LIN {X 0,Y 467.628,Z 314.863,A -85,B 0,C 180,E1 -7719.778,E2 -7719.778} C_VEL
LIN {X 0,Y 467.666,Z 315.024,A -85,B 0,C 180,E1 -7721.055,E2 -7721.055} C_VEL
LIN {X 0,Y 467.97,Z 316.246,A -85,B 0,C 180,E1 -7721.229,E2 -7721.229} C_VEL
LIN {X 0,Y 471.79,Z 327.707,A -85,B 0,C 180,E1 -7721.995,E2 -7721.995} C_VEL
LIN {X 0,Y 471.969,Z 329.737,A -85,B 0,C 180,E1 -7722.115,E2 -7722.115} C_VEL
LIN {X 0,Y 471.397,Z 342.99,A -85,B 0,C 180,E1 -7722.946,E2 -7722.946} C_VEL
LIN {X 0,Y 470.84,Z 354.59,A -85,B 0,C 180,E1 -7723.859,E2 -7723.859} C_VEL
LIN {X 0,Y 470.267,Z 365.932,A -85,B 0,C 180,E1 -7724.95,E2 -7724.95} C_VEL
LIN {X 0,Y 469.698,Z 376.183,A -85,B 0,C 180,E1 -7726.149,E2 -7726.149} C_VEL
LIN {X 0,Y 469.111,Z 385.408,A -85,B 0,C 180,E1 -7727.454,E2 -7727.454} C_VEL
LIN {X 0,Y 468.626,Z 393.041,A -85,B 0,C 180,E1 -7728.758,E2 -7728.758} C_VEL
LIN {X 0,Y 468.253,Z 399.346,A -85,B 0,C 180,E1 -7730.061,E2 -7730.061} C_VEL
LIN {X 0,Y 467.999,Z 404.53,A -85,B 0,C 180,E1 -7731.363,E2 -7731.363} C_VEL
LIN {X 0,Y 467.681,Z 409.923,A -85,B 0,C 180,E1 -7733.095,E2 -7733.095} C_VEL
LIN {X 0,Y 467.396,Z 413.789,A -85,B 0,C 180,E1 -7734.824,E2 -7734.824} C_VEL
LIN {X 0,Y 467.262,Z 416.221,A -85,B 0,C 180,E1 -7736.551,E2 -7736.551} C_VEL
LIN {X 0,Y 467.217,Z 417.297,A -85,B 0,C 180,E1 -7738.276,E2 -7738.276} C_VEL
LIN {X 0,Y 467.122,Z 417.057,A -85,B 0,C 180,E1 -7740,E2 -7740} C_VEL
LIN {X 0,Y 467.22,Z 415.477,A -85,B 0,C 180,E1 -7741.724,E2 -7741.724} C_VEL
LIN {X 0,Y 467.263,Z 412.569,A -85,B 0,C 180,E1 -7743.449,E2 -7743.449} C_VEL
LIN {X 0,Y 467.443,Z 408.228,A -85,B 0,C 180,E1 -7745.176,E2 -7745.176} C_VEL
LIN {X 0,Y 467.782,Z 402.317,A -85,B 0,C 180,E1 -7746.903,E2 -7746.903} C_VEL
LIN {X 0,Y 468.029,Z 395.693,A -85,B 0,C 180,E1 -7748.419,E2 -7748.419} C_VEL
LIN {X 0,Y 468.54,Z 387.434,A -85,B 0,C 180,E1 -7749.933,E2 -7749.933} C_VEL
LIN {X 0,Y 468.977,Z 378.822,A -85,B 0,C 180,E1 -7751.234,E2 -7751.234} C_VEL
LIN {X 0,Y 469.446,Z 370.309,A -85,B 0,C 180,E1 -7752.318,E2 -7752.318} C_VEL
LIN {X 0,Y 470.046,Z 358.967,A -85,B 0,C 180,E1 -7753.521,E2 -7753.521} C_VEL
LIN {X 0,Y 470.599,Z 346.534,A -85,B 0,C 180,E1 -7754.597,E2 -7754.597} C_VEL
LIN {X 0,Y 471.163,Z 334.137,A -85,B 0,C 180,E1 -7755.464,E2 -7755.464} C_VEL
LIN {X 0,Y 471.422,Z 327.577,A -85,B 0,C 180,E1 -7755.851,E2 -7755.851} C_VEL
LIN {X 0,Y 467.73,Z 315.529,A -85,B 0,C 180,E1 -7756.645,E2 -7756.645} C_VEL
LIN {X 0,Y 467.622,Z 314.897,A -85,B 0,C 180,E1 -7756.817,E2 -7756.817} C_VEL
LIN {X 0,Y 467.628,Z 314.862,A -85,B 0,C 180,E1 -7759.308,E2 -7759.308} C_VEL
LIN {X 0,Y 467.539,Z 314.87,A -85,B 0,C 180,E1 -7762.074,E2 -7762.074} C_VEL
LIN {X 0,Y 467.607,Z 314.864,A -85,B 0,C 180,E1 -7764.887,E2 -7764.887} C_VEL
LIN {X 0,Y 467.625,Z 314.856,A -85,B 0,C 180,E1 -7767.769,E2 -7767.769} C_VEL
LIN {X 0,Y 467.573,Z 314.865,A -85,B 0,C 180,E1 -7771.045,E2 -7771.045} C_VEL
LIN {X 0,Y 467.595,Z 314.863,A -85,B 0,C 180,E1 -7774.243,E2 -7774.243} C_VEL
LIN {X 0,Y 467.555,Z 314.866,A -85,B 0,C 180,E1 -7777.187,E2 -7777.187} C_VEL
LIN {X 0,Y 467.58,Z 314.867,A -85,B 0,C 180,E1 -7780.265,E2 -7780.265} C_VEL
LIN {X 0,Y 467.592,Z 314.867,A -85,B 0,C 180,E1 -7782.567,E2 -7782.567} C_VEL
LIN {X 0,Y 467.576,Z 314.863,A -85,B 0,C 180,E1 -7785.053,E2 -7785.053} C_VEL
LIN {X 0,Y 467.594,Z 314.86,A -85,B 0,C 180,E1 -7787.44,E2 -7787.44} C_VEL
LIN {X 0,Y 467.588,Z 314.863,A -85,B 0,C 180,E1 -7790.855,E2 -7790.855} C_VEL
LIN {X 0,Y 467.565,Z 314.872,A -85,B 0,C 180,E1 -7794.261,E2 -7794.261} C_VEL
LIN {X 0,Y 467.588,Z 314.861,A -85,B 0,C 180,E1 -7797.321,E2 -7797.321} C_VEL
LIN {X 0,Y 467.576,Z 314.864,A -85,B 0,C 180,E1 -7800.667,E2 -7800.667} C_VEL
LIN {X 0,Y 467.619,Z 314.857,A -85,B 0,C 180,E1 -7803.199,E2 -7803.199} C_VEL
LIN {X 0,Y 467.597,Z 314.863,A -85,B 0,C 180,E1 -7806.468,E2 -7806.468} C_VEL
LIN {X 0,Y 467.629,Z 314.86,A -85,B 0,C 180,E1 -7809.777,E2 -7809.777} C_VEL
LIN {X 0,Y 467.618,Z 314.857,A -85,B 0,C 180,E1 -7810.433,E2 -7810.433} C_VEL
LIN {X 0,Y 466.981,Z 314.938,A -85,B 0,C 180,E1 -7811.152,E2 -7811.152} C_VEL
LIN {X 0,Y 464.166,Z 315.296,A -85,B 0,C 180,E1 -7812.319,E2 -7812.319} C_VEL
LIN {X 0,Y 461.754,Z 315.599,A -85,B 0,C 180,E1 -7813.26,E2 -7813.26} C_VEL
LIN {X 0,Y 460.693,Z 315.728,A -85,B 0,C 180,E1 -7813.987,E2 -7813.987} C_VEL
LIN {X 0,Y 460.594,Z 315.737,A -85,B 0,C 180,E1 -7814.233,E2 -7814.233} C_VEL
LIN {X 0,Y 460.615,Z 315.734,A -85,B 0,C 180,E1 -7817.665,E2 -7817.665} C_VEL
LIN {X 0,Y 460.633,Z 315.728,A -85,B 0,C 180,E1 -7821.223,E2 -7821.223} C_VEL
LIN {X 0,Y 460.707,Z 315.726,A -85,B 0,C 180,E1 -7823.869,E2 -7823.869} C_VEL
LIN {X 0,Y 460.805,Z 315.708,A -85,B 0,C 180,E1 -7827.377,E2 -7827.377} C_VEL
LIN {X 0,Y 460.858,Z 315.704,A -85,B 0,C 180,E1 -7829.999,E2 -7829.999} C_VEL
LIN {X 0,Y 460.805,Z 315.706,A -85,B 0,C 180,E1 -7832.622,E2 -7832.622} C_VEL
LIN {X 0,Y 460.714,Z 315.719,A -85,B 0,C 180,E1 -7836.129,E2 -7836.129} C_VEL
LIN {X 0,Y 460.633,Z 315.727,A -85,B 0,C 180,E1 -7838.775,E2 -7838.775} C_VEL
LIN {X 0,Y 460.617,Z 315.729,A -85,B 0,C 180,E1 -7842.444,E2 -7842.444} C_VEL
LIN {X 0,Y 460.603,Z 315.733,A -85,B 0,C 180,E1 -7845.996,E2 -7845.996} C_VEL
LIN {X 0,Y 460.574,Z 315.736,A -85,B 0,C 180,E1 -7848.901,E2 -7848.901} C_VEL
LIN {X 0,Y 460.518,Z 315.749,A -85,B 0,C 180,E1 -7851.484,E2 -7851.484} C_VEL
LIN {X 0,Y 460.544,Z 315.738,A -85,B 0,C 180,E1 -7854.331,E2 -7854.331} C_VEL
LIN {X 0,Y 460.58,Z 315.741,A -85,B 0,C 180,E1 -7857.242,E2 -7857.242} C_VEL
LIN {X 0,Y 460.511,Z 315.742,A -85,B 0,C 180,E1 -7860.239,E2 -7860.239} C_VEL
LIN {X 0,Y 460.528,Z 315.747,A -85,B 0,C 180,E1 -7863.324,E2 -7863.324} C_VEL
LIN {X 0,Y 460.475,Z 315.748,A -85,B 0,C 180,E1 -7866.528,E2 -7866.528} C_VEL
LIN {X 0,Y 460.531,Z 315.74,A -85,B 0,C 180,E1 -7869.861,E2 -7869.861} C_VEL
LIN {X 0,Y 460.514,Z 315.747,A -85,B 0,C 180,E1 -7872.9,E2 -7872.9} C_VEL
LIN {X 0,Y 460.517,Z 315.742,A -85,B 0,C 180,E1 -7875.828,E2 -7875.828} C_VEL
LIN {X 0,Y 460.527,Z 315.748,A -85,B 0,C 180,E1 -7878.988,E2 -7878.988} C_VEL
LIN {X 0,Y 460.528,Z 315.744,A -85,B 0,C 180,E1 -7881.267,E2 -7881.267} C_VEL
LIN {X 0,Y 460.509,Z 315.746,A -85,B 0,C 180,E1 -7884.554,E2 -7884.554} C_VEL
LIN {X 0,Y 460.528,Z 315.74,A -85,B 0,C 180,E1 -7887.715,E2 -7887.715} C_VEL
LIN {X 0,Y 460.543,Z 315.746,A -85,B 0,C 180,E1 -7890.769,E2 -7890.769} C_VEL
LIN {X 0,Y 460.562,Z 315.736,A -85,B 0,C 180,E1 -7893.734,E2 -7893.734} C_VEL
LIN {X 0,Y 460.54,Z 315.745,A -85,B 0,C 180,E1 -7896.623,E2 -7896.623} C_VEL
LIN {X 0,Y 460.545,Z 315.738,A -85,B 0,C 180,E1 -7899.452,E2 -7899.452} C_VEL
LIN {X 0,Y 460.553,Z 315.74,A -85,B 0,C 180,E1 -7902.23,E2 -7902.23} C_VEL
LIN {X 0,Y 460.558,Z 315.74,A -85,B 0,C 180,E1 -7904.964,E2 -7904.964} C_VEL
LIN {X 0,Y 460.604,Z 315.739,A -85,B 0,C 180,E1 -7908.559,E2 -7908.559} C_VEL
LIN {X 0,Y 460.687,Z 315.723,A -85,B 0,C 180,E1 -7912.108,E2 -7912.108} C_VEL
LIN {X 0,Y 460.691,Z 315.724,A -85,B 0,C 180,E1 -7914.748,E2 -7914.748} C_VEL
LIN {X 0,Y 460.818,Z 315.704,A -85,B 0,C 180,E1 -7917.377,E2 -7917.377} C_VEL
LIN {X 0,Y 460.845,Z 315.704,A -85,B 0,C 180,E1 -7920,E2 -7920} C_VEL
LIN {X 0,Y 460.818,Z 315.708,A -85,B 0,C 180,E1 -7922.622,E2 -7922.622} C_VEL
LIN {X 0,Y 460.702,Z 315.724,A -85,B 0,C 180,E1 -7926.13,E2 -7926.13} C_VEL
LIN {X 0,Y 460.621,Z 315.73,A -85,B 0,C 180,E1 -7928.776,E2 -7928.776} C_VEL
LIN {X 0,Y 460.626,Z 315.732,A -85,B 0,C 180,E1 -7932.457,E2 -7932.457} C_VEL
LIN {X 0,Y 460.613,Z 315.736,A -85,B 0,C 180,E1 -7936.007,E2 -7936.007} C_VEL
LIN {X 0,Y 460.561,Z 315.738,A -85,B 0,C 180,E1 -7939.616,E2 -7939.616} C_VEL
LIN {X 0,Y 460.505,Z 315.746,A -85,B 0,C 180,E1 -7942.429,E2 -7942.429} C_VEL
LIN {X 0,Y 460.56,Z 315.742,A -85,B 0,C 180,E1 -7945.802,E2 -7945.802} C_VEL
LIN {X 0,Y 460.551,Z 315.742,A -85,B 0,C 180,E1 -7948.233,E2 -7948.233} C_VEL
LIN {X 0,Y 460.518,Z 315.742,A -85,B 0,C 180,E1 -7951.284,E2 -7951.284} C_VEL
LIN {X 0,Y 460.527,Z 315.741,A -85,B 0,C 180,E1 -7954.507,E2 -7954.507} C_VEL
LIN {X 0,Y 460.524,Z 315.748,A -85,B 0,C 180,E1 -7957.621,E2 -7957.621} C_VEL
LIN {X 0,Y 460.553,Z 315.743,A -85,B 0,C 180,E1 -7960.273,E2 -7960.273} C_VEL
LIN {X 0,Y 460.494,Z 315.751,A -85,B 0,C 180,E1 -7963.376,E2 -7963.376} C_VEL
LIN {X 0,Y 460.581,Z 315.992,A -85,B 0,C 180,E1 -7965.106,E2 -7965.106} C_VEL
LIN {X 0,Y 462.621,Z 325.576,A -85,B 0,C 180,E1 -7968.107,E2 -7968.107} C_VEL
LIN {X 0,Y 464.108,Z 333.816,A -85,B 0,C 180,E1 -7970.56,E2 -7970.56} C_VEL
LIN {X 0,Y 463.807,Z 340.288,A -85,B 0,C 180,E1 -7972.33,E2 -7972.33} C_VEL
LIN {X 0,Y 462.916,Z 353.475,A -85,B 0,C 180,E1 -7975.825,E2 -7975.825} C_VEL
LIN {X 0,Y 462.307,Z 365.318,A -85,B 0,C 180,E1 -7978.879,E2 -7978.879} C_VEL
LIN {X 0,Y 461.866,Z 375.16,A -85,B 0,C 180,E1 -7981.36,E2 -7981.36} C_VEL
LIN {X 0,Y 461.397,Z 387.321,A -85,B 0,C 180,E1 -7984.365,E2 -7984.365} C_VEL
LIN {X 0,Y 461.011,Z 398.687,A -85,B 0,C 180,E1 -7987.125,E2 -7987.125} C_VEL
LIN {X 0,Y 460.583,Z 412.328,A -85,B 0,C 180,E1 -7990.386,E2 -7990.386} C_VEL
LIN {X 0,Y 460.517,Z 415.483,A -85,B 0,C 180,E1 -7991.083,E2 -7991.083} C_VEL
LIN {X 0,Y 461.15,Z 420.195,A -85,B 0,C 180,E1 -7991.244,E2 -7991.244} C_VEL
LIN {X 0,Y 462.995,Z 434.142,A -85,B 0,C 180,E1 -7991.685,E2 -7991.685} C_VEL
LIN {X 0,Y 464.3,Z 444.091,A -85,B 0,C 180,E1 -7992.094,E2 -7992.094} C_VEL
LIN {X 0,Y 463.679,Z 457.656,A -85,B 0,C 180,E1 -7992.725,E2 -7992.725} C_VEL
LIN {X 0,Y 462.956,Z 471.604,A -85,B 0,C 180,E1 -7993.577,E2 -7993.577} C_VEL
LIN {X 0,Y 462.209,Z 484.511,A -85,B 0,C 180,E1 -7994.569,E2 -7994.569} C_VEL
LIN {X 0,Y 461.577,Z 496.243,A -85,B 0,C 180,E1 -7995.676,E2 -7995.676} C_VEL
LIN {X 0,Y 460.939,Z 507.823,A -85,B 0,C 180,E1 -7997.004,E2 -7997.004} C_VEL
LIN {X 0,Y 460.56,Z 517.359,A -85,B 0,C 180,E1 -7998.336,E2 -7998.336} C_VEL
LIN {X 0,Y 460.142,Z 526.442,A -85,B 0,C 180,E1 -7999.885,E2 -7999.885} C_VEL
LIN {X 0,Y 459.972,Z 532.875,A -85,B 0,C 180,E1 -8001.212,E2 -8001.212} C_VEL
LIN {X 0,Y 459.892,Z 538.158,A -85,B 0,C 180,E1 -8002.537,E2 -8002.537} C_VEL
LIN {X 0,Y 459.93,Z 542.435,A -85,B 0,C 180,E1 -8003.861,E2 -8003.861} C_VEL
LIN {X 0,Y 459.886,Z 546.709,A -85,B 0,C 180,E1 -8005.619,E2 -8005.619} C_VEL
LIN {X 0,Y 459.897,Z 549.469,A -85,B 0,C 180,E1 -8007.373,E2 -8007.373} C_VEL
LIN {X 0,Y 459.864,Z 550.771,A -85,B 0,C 180,E1 -8009.125,E2 -8009.125} C_VEL
LIN {X 0,Y 459.999,Z 550.906,A -85,B 0,C 180,E1 -8010.001,E2 -8010.001} C_VEL
LIN {X 0,Y 460.019,Z 550.665,A -85,B 0,C 180,E1 -8010.876,E2 -8010.876} C_VEL
LIN {X 0,Y 459.945,Z 549.078,A -85,B 0,C 180,E1 -8012.628,E2 -8012.628} C_VEL
LIN {X 0,Y 460.043,Z 546.043,A -85,B 0,C 180,E1 -8014.382,E2 -8014.382} C_VEL
LIN {X 0,Y 459.977,Z 542.746,A -85,B 0,C 180,E1 -8015.7,E2 -8015.7} C_VEL
LIN {X 0,Y 460.012,Z 536.886,A -85,B 0,C 180,E1 -8017.462,E2 -8017.462} C_VEL
LIN {X 0,Y 460.066,Z 530.243,A -85,B 0,C 180,E1 -8019.009,E2 -8019.009} C_VEL
LIN {X 0,Y 460.301,Z 521.996,A -85,B 0,C 180,E1 -8020.558,E2 -8020.558} C_VEL
LIN {X 0,Y 460.556,Z 513.41,A -85,B 0,C 180,E1 -8021.889,E2 -8021.889} C_VEL
LIN {X 0,Y 460.958,Z 503.141,A -85,B 0,C 180,E1 -8023.221,E2 -8023.221} C_VEL
LIN {X 0,Y 461.475,Z 491.831,A -85,B 0,C 180,E1 -8024.442,E2 -8024.442} C_VEL
LIN {X 0,Y 462.189,Z 479.47,A -85,B 0,C 180,E1 -8025.546,E2 -8025.546} C_VEL
LIN {X 0,Y 462.842,Z 465.889,A -85,B 0,C 180,E1 -8026.542,E2 -8026.542} C_VEL
LIN {X 0,Y 463.548,Z 452.57,A -85,B 0,C 180,E1 -8027.319,E2 -8027.319} C_VEL
LIN {X 0,Y 463.934,Z 443.508,A -85,B 0,C 180,E1 -8027.751,E2 -8027.751} C_VEL
LIN {X 0,Y 462.67,Z 432.253,A -85,B 0,C 180,E1 -8028.259,E2 -8028.259} C_VEL
LIN {X 0,Y 461.343,Z 416.975,A -85,B 0,C 180,E1 -8028.776,E2 -8028.776} C_VEL
LIN {X 0,Y 460.379,Z 409.518,A -85,B 0,C 180,E1 -8029.018,E2 -8029.018} C_VEL
LIN {X 0,Y 460.435,Z 407.458,A -85,B 0,C 180,E1 -8029.395,E2 -8029.395} C_VEL
LIN {X 0,Y 460.579,Z 392.689,A -85,B 0,C 180,E1 -8032.662,E2 -8032.662} C_VEL
LIN {X 0,Y 460.751,Z 378.539,A -85,B 0,C 180,E1 -8035.849,E2 -8035.849} C_VEL
LIN {X 0,Y 460.983,Z 364.098,A -85,B 0,C 180,E1 -8039.201,E2 -8039.201} C_VEL
LIN {X 0,Y 461.17,Z 351.605,A -85,B 0,C 180,E1 -8042.235,E2 -8042.235} C_VEL
LIN {X 0,Y 461.757,Z 337.842,A -85,B 0,C 180,E1 -8045.8,E2 -8045.8} C_VEL
LIN {X 0,Y 462.679,Z 328.181,A -85,B 0,C 180,E1 -8048.52,E2 -8048.52} C_VEL
LIN {X 0,Y 462.076,Z 323.427,A -85,B 0,C 180,E1 -8050.069,E2 -8050.069} C_VEL
LIN {X 0,Y 460.965,Z 317.845,A -85,B 0,C 180,E1 -8052.132,E2 -8052.132} C_VEL
LIN {X 0,Y 460.532,Z 315.801,A -85,B 0,C 180,E1 -8052.999,E2 -8052.999} C_VEL
LIN {X 0,Y 460.515,Z 315.749,A -85,B 0,C 180,E1 -8055.831,E2 -8055.831} C_VEL
LIN {X 0,Y 460.542,Z 315.744,A -85,B 0,C 180,E1 -8058.99,E2 -8058.99} C_VEL
LIN {X 0,Y 460.547,Z 315.744,A -85,B 0,C 180,E1 -8061.269,E2 -8061.269} C_VEL
LIN {X 0,Y 460.517,Z 315.744,A -85,B 0,C 180,E1 -8064.555,E2 -8064.555} C_VEL
LIN {X 0,Y 460.535,Z 315.746,A -85,B 0,C 180,E1 -8067.716,E2 -8067.716} C_VEL
LIN {X 0,Y 460.543,Z 315.742,A -85,B 0,C 180,E1 -8070.769,E2 -8070.769} C_VEL
LIN {X 0,Y 460.567,Z 315.741,A -85,B 0,C 180,E1 -8073.735,E2 -8073.735} C_VEL
LIN {X 0,Y 460.55,Z 315.743,A -85,B 0,C 180,E1 -8076.624,E2 -8076.624} C_VEL
LIN {X 0,Y 460.556,Z 315.744,A -85,B 0,C 180,E1 -8079.453,E2 -8079.453} C_VEL
LIN {X 0,Y 460.633,Z 315.941,A -85,B 0,C 180,E1 -8080.733,E2 -8080.733} C_VEL
LIN {X 0,Y 460.904,Z 317.05,A -85,B 0,C 180,E1 -8080.892,E2 -8080.892} C_VEL
LIN {X 0,Y 465.016,Z 329.082,A -85,B 0,C 180,E1 -8081.724,E2 -8081.724} C_VEL
LIN {X 0,Y 465.252,Z 332.956,A -85,B 0,C 180,E1 -8081.961,E2 -8081.961} C_VEL
LIN {X 0,Y 464.64,Z 345.545,A -85,B 0,C 180,E1 -8082.791,E2 -8082.791} C_VEL
LIN {X 0,Y 464.029,Z 358.222,A -85,B 0,C 180,E1 -8083.841,E2 -8083.841} C_VEL
LIN {X 0,Y 463.39,Z 369.118,A -85,B 0,C 180,E1 -8084.946,E2 -8084.946} C_VEL
LIN {X 0,Y 462.771,Z 379.447,A -85,B 0,C 180,E1 -8086.221,E2 -8086.221} C_VEL
LIN {X 0,Y 462.228,Z 387.925,A -85,B 0,C 180,E1 -8087.487,E2 -8087.487} C_VEL
LIN {X 0,Y 461.586,Z 396.39,A -85,B 0,C 180,E1 -8089.029,E2 -8089.029} C_VEL
LIN {X 0,Y 461.197,Z 402.314,A -85,B 0,C 180,E1 -8090.35,E2 -8090.35} C_VEL
LIN {X 0,Y 460.937,Z 407.14,A -85,B 0,C 180,E1 -8091.672,E2 -8091.672} C_VEL
LIN {X 0,Y 460.681,Z 412.123,A -85,B 0,C 180,E1 -8093.43,E2 -8093.43} C_VEL
LIN {X 0,Y 460.404,Z 414.86,A -85,B 0,C 180,E1 -8094.745,E2 -8094.745} C_VEL
LIN {X 0,Y 460.25,Z 417.278,A -85,B 0,C 180,E1 -8096.498,E2 -8096.498} C_VEL
LIN {X 0,Y 460.201,Z 418.341,A -85,B 0,C 180,E1 -8098.25,E2 -8098.25} C_VEL
LIN {X 0,Y 460.1,Z 418.084,A -85,B 0,C 180,E1 -8100,E2 -8100} C_VEL
LIN {X 0,Y 460.203,Z 416.483,A -85,B 0,C 180,E1 -8101.75,E2 -8101.75} C_VEL
LIN {X 0,Y 460.244,Z 413.549,A -85,B 0,C 180,E1 -8103.502,E2 -8103.502} C_VEL
LIN {X 0,Y 460.443,Z 409.175,A -85,B 0,C 180,E1 -8105.255,E2 -8105.255} C_VEL
LIN {X 0,Y 460.806,Z 403.228,A -85,B 0,C 180,E1 -8107.009,E2 -8107.009} C_VEL
LIN {X 0,Y 461.078,Z 396.57,A -85,B 0,C 180,E1 -8108.547,E2 -8108.547} C_VEL
LIN {X 0,Y 461.612,Z 388.269,A -85,B 0,C 180,E1 -8110.084,E2 -8110.084} C_VEL
LIN {X 0,Y 462.074,Z 379.621,A -85,B 0,C 180,E1 -8111.404,E2 -8111.404} C_VEL
LIN {X 0,Y 462.574,Z 371.079,A -85,B 0,C 180,E1 -8112.504,E2 -8112.504} C_VEL
LIN {X 0,Y 463.192,Z 359.827,A -85,B 0,C 180,E1 -8113.711,E2 -8113.711} C_VEL
LIN {X 0,Y 463.728,Z 348.623,A -85,B 0,C 180,E1 -8114.706,E2 -8114.706} C_VEL
LIN {X 0,Y 464.356,Z 336.506,A -85,B 0,C 180,E1 -8115.584,E2 -8115.584} C_VEL
LIN {X 0,Y 464.596,Z 328.994,A -85,B 0,C 180,E1 -8116.045,E2 -8116.045} C_VEL
LIN {X 0,Y 460.652,Z 316.238,A -85,B 0,C 180,E1 -8116.908,E2 -8116.908} C_VEL
LIN {X 0,Y 460.591,Z 315.767,A -85,B 0,C 180,E1 -8117.082,E2 -8117.082} C_VEL
LIN {X 0,Y 460.573,Z 315.739,A -85,B 0,C 180,E1 -8119.616,E2 -8119.616} C_VEL
LIN {X 0,Y 460.515,Z 315.748,A -85,B 0,C 180,E1 -8122.429,E2 -8122.429} C_VEL
LIN {X 0,Y 460.573,Z 315.734,A -85,B 0,C 180,E1 -8125.802,E2 -8125.802} C_VEL
LIN {X 0,Y 460.557,Z 315.739,A -85,B 0,C 180,E1 -8128.233,E2 -8128.233} C_VEL
LIN {X 0,Y 460.526,Z 315.741,A -85,B 0,C 180,E1 -8131.283,E2 -8131.283} C_VEL
LIN {X 0,Y 460.539,Z 315.746,A -85,B 0,C 180,E1 -8134.506,E2 -8134.506} C_VEL
LIN {X 0,Y 460.507,Z 315.743,A -85,B 0,C 180,E1 -8137.623,E2 -8137.623} C_VEL
LIN {X 0,Y 460.544,Z 315.743,A -85,B 0,C 180,E1 -8140.269,E2 -8140.269} C_VEL
LIN {X 0,Y 460.503,Z 315.743,A -85,B 0,C 180,E1 -8143.376,E2 -8143.376} C_VEL
LIN {X 0,Y 460.515,Z 315.747,A -85,B 0,C 180,E1 -8146.626,E2 -8146.626} C_VEL
LIN {X 0,Y 460.549,Z 315.739,A -85,B 0,C 180,E1 -8149.73,E2 -8149.73} C_VEL
LIN {X 0,Y 460.505,Z 315.748,A -85,B 0,C 180,E1 -8152.524,E2 -8152.524} C_VEL
LIN {X 0,Y 460.552,Z 315.738,A -85,B 0,C 180,E1 -8155.624,E2 -8155.624} C_VEL
LIN {X 0,Y 460.543,Z 315.74,A -85,B 0,C 180,E1 -8158.744,E2 -8158.744} C_VEL
LIN {X 0,Y 460.595,Z 315.739,A -85,B 0,C 180,E1 -8162.252,E2 -8162.252} C_VEL
LIN {X 0,Y 460.538,Z 315.741,A -85,B 0,C 180,E1 -8165.667,E2 -8165.667} C_VEL
LIN {X 0,Y 460.528,Z 315.742,A -85,B 0,C 180,E1 -8168.578,E2 -8168.578} C_VEL
LIN {X 0,Y 460.597,Z 315.732,A -85,B 0,C 180,E1 -8171.311,E2 -8171.311} C_VEL
LIN {X 0,Y 460.594,Z 315.737,A -85,B 0,C 180,E1 -8174.233,E2 -8174.233} C_VEL
LIN {X 0,Y 459.892,Z 315.82,A -85,B 0,C 180,E1 -8174.963,E2 -8174.963} C_VEL
LIN {X 0,Y 457.031,Z 316.181,A -85,B 0,C 180,E1 -8176.148,E2 -8176.148} C_VEL
LIN {X 0,Y 454.642,Z 316.476,A -85,B 0,C 180,E1 -8177.104,E2 -8177.104} C_VEL
LIN {X 0,Y 453.631,Z 316.606,A -85,B 0,C 180,E1 -8177.842,E2 -8177.842} C_VEL
LIN {X 0,Y 453.555,Z 316.61,A -85,B 0,C 180,E1 -8178.092,E2 -8178.092} C_VEL
LIN {X 0,Y 453.597,Z 316.604,A -85,B 0,C 180,E1 -8181.086,E2 -8181.086} C_VEL
LIN {X 0,Y 453.675,Z 316.601,A -85,B 0,C 180,E1 -8183.774,E2 -8183.774} C_VEL
LIN {X 0,Y 453.749,Z 316.587,A -85,B 0,C 180,E1 -8187.336,E2 -8187.336} C_VEL
LIN {X 0,Y 453.828,Z 316.579,A -85,B 0,C 180,E1 -8189.999,E2 -8189.999} C_VEL
LIN {X 0,Y 453.749,Z 316.584,A -85,B 0,C 180,E1 -8192.662,E2 -8192.662} C_VEL
LIN {X 0,Y 453.682,Z 316.594,A -85,B 0,C 180,E1 -8196.224,E2 -8196.224} C_VEL
LIN {X 0,Y 453.596,Z 316.604,A -85,B 0,C 180,E1 -8198.912,E2 -8198.912} C_VEL
LIN {X 0,Y 453.567,Z 316.607,A -85,B 0,C 180,E1 -8202.528,E2 -8202.528} C_VEL
LIN {X 0,Y 453.548,Z 316.61,A -85,B 0,C 180,E1 -8206.195,E2 -8206.195} C_VEL
LIN {X 0,Y 453.523,Z 316.615,A -85,B 0,C 180,E1 -8209.04,E2 -8209.04} C_VEL
LIN {X 0,Y 453.479,Z 316.621,A -85,B 0,C 180,E1 -8211.835,E2 -8211.835} C_VEL
LIN {X 0,Y 453.515,Z 316.615,A -85,B 0,C 180,E1 -8214.733,E2 -8214.733} C_VEL
LIN {X 0,Y 453.538,Z 316.612,A -85,B 0,C 180,E1 -8217.96,E2 -8217.96} C_VEL
LIN {X 0,Y 453.467,Z 316.624,A -85,B 0,C 180,E1 -8221.524,E2 -8221.524} C_VEL
LIN {X 0,Y 453.486,Z 316.62,A -85,B 0,C 180,E1 -8224.776,E2 -8224.776} C_VEL
LIN {X 0,Y 453.463,Z 316.62,A -85,B 0,C 180,E1 -8228.31,E2 -8228.31} C_VEL
LIN {X 0,Y 453.492,Z 316.618,A -85,B 0,C 180,E1 -8230.608,E2 -8230.608} C_VEL
LIN {X 0,Y 453.461,Z 316.626,A -85,B 0,C 180,E1 -8233.244,E2 -8233.244} C_VEL
LIN {X 0,Y 453.471,Z 316.62,A -85,B 0,C 180,E1 -8235.779,E2 -8235.779} C_VEL
LIN {X 0,Y 453.49,Z 316.62,A -85,B 0,C 180,E1 -8239.39,E2 -8239.39} C_VEL
LIN {X 0,Y 453.47,Z 316.62,A -85,B 0,C 180,E1 -8242.222,E2 -8242.222} C_VEL
LIN {X 0,Y 453.484,Z 316.621,A -85,B 0,C 180,E1 -8245.221,E2 -8245.221} C_VEL
LIN {X 0,Y 453.482,Z 316.621,A -85,B 0,C 180,E1 -8248.469,E2 -8248.469} C_VEL
LIN {X 0,Y 453.51,Z 316.617,A -85,B 0,C 180,E1 -8251.288,E2 -8251.288} C_VEL
LIN {X 0,Y 453.519,Z 316.615,A -85,B 0,C 180,E1 -8254.284,E2 -8254.284} C_VEL
LIN {X 0,Y 453.474,Z 316.621,A -85,B 0,C 180,E1 -8257.203,E2 -8257.203} C_VEL
LIN {X 0,Y 453.498,Z 316.617,A -85,B 0,C 180,E1 -8260.065,E2 -8260.065} C_VEL
LIN {X 0,Y 453.5,Z 316.62,A -85,B 0,C 180,E1 -8262.875,E2 -8262.875} C_VEL
LIN {X 0,Y 453.508,Z 316.614,A -85,B 0,C 180,E1 -8265.643,E2 -8265.643} C_VEL
LIN {X 0,Y 453.552,Z 316.615,A -85,B 0,C 180,E1 -8268.378,E2 -8268.378} C_VEL
LIN {X 0,Y 453.644,Z 316.6,A -85,B 0,C 180,E1 -8271.985,E2 -8271.985} C_VEL
LIN {X 0,Y 453.664,Z 316.6,A -85,B 0,C 180,E1 -8274.666,E2 -8274.666} C_VEL
LIN {X 0,Y 453.759,Z 316.583,A -85,B 0,C 180,E1 -8277.337,E2 -8277.337} C_VEL
LIN {X 0,Y 453.815,Z 316.579,A -85,B 0,C 180,E1 -8280,E2 -8280} C_VEL
LIN {X 0,Y 453.758,Z 316.587,A -85,B 0,C 180,E1 -8282.663,E2 -8282.663} C_VEL
LIN {X 0,Y 453.669,Z 316.602,A -85,B 0,C 180,E1 -8286.225,E2 -8286.225} C_VEL
LIN {X 0,Y 453.585,Z 316.606,A -85,B 0,C 180,E1 -8288.913,E2 -8288.913} C_VEL
LIN {X 0,Y 453.593,Z 316.607,A -85,B 0,C 180,E1 -8292.551,E2 -8292.551} C_VEL
LIN {X 0,Y 453.548,Z 316.617,A -85,B 0,C 180,E1 -8296.196,E2 -8296.196} C_VEL
LIN {X 0,Y 453.512,Z 316.614,A -85,B 0,C 180,E1 -8299.041,E2 -8299.041} C_VEL
LIN {X 0,Y 453.469,Z 316.625,A -85,B 0,C 180,E1 -8301.836,E2 -8301.836} C_VEL
LIN {X 0,Y 453.506,Z 316.615,A -85,B 0,C 180,E1 -8304.735,E2 -8304.735} C_VEL
LIN {X 0,Y 453.531,Z 316.62,A -85,B 0,C 180,E1 -8307.962,E2 -8307.962} C_VEL
LIN {X 0,Y 453.476,Z 316.619,A -85,B 0,C 180,E1 -8310.759,E2 -8310.759} C_VEL
LIN {X 0,Y 453.471,Z 316.627,A -85,B 0,C 180,E1 -8313.913,E2 -8313.913} C_VEL
LIN {X 0,Y 453.465,Z 316.624,A -85,B 0,C 180,E1 -8317.188,E2 -8317.188} C_VEL
LIN {X 0,Y 453.527,Z 316.619,A -85,B 0,C 180,E1 -8319.446,E2 -8319.446} C_VEL
LIN {X 0,Y 453.457,Z 316.627,A -85,B 0,C 180,E1 -8322.996,E2 -8322.996} C_VEL
LIN {X 0,Y 453.502,Z 316.721,A -85,B 0,C 180,E1 -8324.704,E2 -8324.704} C_VEL
LIN {X 0,Y 455.774,Z 327.457,A -85,B 0,C 180,E1 -8328.133,E2 -8328.133} C_VEL
LIN {X 0,Y 457.078,Z 334.436,A -85,B 0,C 180,E1 -8330.246,E2 -8330.246} C_VEL
LIN {X 0,Y 457.067,Z 339.38,A -85,B 0,C 180,E1 -8331.646,E2 -8331.646} C_VEL
LIN {X 0,Y 456.085,Z 352.675,A -85,B 0,C 180,E1 -8335.241,E2 -8335.241} C_VEL
LIN {X 0,Y 455.287,Z 366.482,A -85,B 0,C 180,E1 -8338.862,E2 -8338.862} C_VEL
LIN {X 0,Y 454.746,Z 377.777,A -85,B 0,C 180,E1 -8341.754,E2 -8341.754} C_VEL
LIN {X 0,Y 454.26,Z 390.027,A -85,B 0,C 180,E1 -8344.821,E2 -8344.821} C_VEL
LIN {X 0,Y 453.842,Z 401.744,A -85,B 0,C 180,E1 -8347.705,E2 -8347.705} C_VEL
LIN {X 0,Y 453.476,Z 414.662,A -85,B 0,C 180,E1 -8350.793,E2 -8350.793} C_VEL
LIN {X 0,Y 453.922,Z 418.365,A -85,B 0,C 180,E1 -8350.934,E2 -8350.934} C_VEL
LIN {X 0,Y 455.929,Z 433.006,A -85,B 0,C 180,E1 -8351.405,E2 -8351.405} C_VEL
LIN {X 0,Y 457.371,Z 445.321,A -85,B 0,C 180,E1 -8351.93,E2 -8351.93} C_VEL
LIN {X 0,Y 456.694,Z 459.444,A -85,B 0,C 180,E1 -8352.635,E2 -8352.635} C_VEL
LIN {X 0,Y 455.973,Z 471.938,A -85,B 0,C 180,E1 -8353.434,E2 -8353.434} C_VEL
LIN {X 0,Y 455.204,Z 484.622,A -85,B 0,C 180,E1 -8354.44,E2 -8354.44} C_VEL
LIN {X 0,Y 454.543,Z 496.182,A -85,B 0,C 180,E1 -8355.564,E2 -8355.564} C_VEL
LIN {X 0,Y 453.905,Z 506.719,A -85,B 0,C 180,E1 -8356.799,E2 -8356.799} C_VEL
LIN {X 0,Y 453.527,Z 516.313,A -85,B 0,C 180,E1 -8358.154,E2 -8358.154} C_VEL
LIN {X 0,Y 453.107,Z 525.417,A -85,B 0,C 180,E1 -8359.726,E2 -8359.726} C_VEL
LIN {X 0,Y 452.918,Z 531.862,A -85,B 0,C 180,E1 -8361.074,E2 -8361.074} C_VEL
LIN {X 0,Y 452.824,Z 537.147,A -85,B 0,C 180,E1 -8362.42,E2 -8362.42} C_VEL
LIN {X 0,Y 452.878,Z 541.438,A -85,B 0,C 180,E1 -8363.765,E2 -8363.765} C_VEL
LIN {X 0,Y 452.836,Z 545.715,A -85,B 0,C 180,E1 -8365.55,E2 -8365.55} C_VEL
LIN {X 0,Y 452.855,Z 548.473,A -85,B 0,C 180,E1 -8367.332,E2 -8367.332} C_VEL
LIN {X 0,Y 452.834,Z 549.77,A -85,B 0,C 180,E1 -8369.112,E2 -8369.112} C_VEL
LIN {X 0,Y 452.982,Z 549.902,A -85,B 0,C 180,E1 -8370.001,E2 -8370.001} C_VEL
LIN {X 0,Y 453.002,Z 549.652,A -85,B 0,C 180,E1 -8370.89,E2 -8370.89} C_VEL
LIN {X 0,Y 452.908,Z 548.041,A -85,B 0,C 180,E1 -8372.669,E2 -8372.669} C_VEL
LIN {X 0,Y 453.017,Z 544.977,A -85,B 0,C 180,E1 -8374.45,E2 -8374.45} C_VEL
LIN {X 0,Y 452.931,Z 540.324,A -85,B 0,C 180,E1 -8376.236,E2 -8376.236} C_VEL
LIN {X 0,Y 452.949,Z 535.758,A -85,B 0,C 180,E1 -8377.579,E2 -8377.579} C_VEL
LIN {X 0,Y 453.02,Z 529.079,A -85,B 0,C 180,E1 -8379.15,E2 -8379.15} C_VEL
LIN {X 0,Y 453.222,Z 520.794,A -85,B 0,C 180,E1 -8380.725,E2 -8380.725} C_VEL
LIN {X 0,Y 453.488,Z 511.168,A -85,B 0,C 180,E1 -8382.222,E2 -8382.222} C_VEL
LIN {X 0,Y 454.055,Z 500.016,A -85,B 0,C 180,E1 -8383.654,E2 -8383.654} C_VEL
LIN {X 0,Y 454.617,Z 488.348,A -85,B 0,C 180,E1 -8384.893,E2 -8384.893} C_VEL
LIN {X 0,Y 455.364,Z 475.478,A -85,B 0,C 180,E1 -8386.015,E2 -8386.015} C_VEL
LIN {X 0,Y 456.091,Z 462.998,A -85,B 0,C 180,E1 -8386.909,E2 -8386.909} C_VEL
LIN {X 0,Y 456.861,Z 448.806,A -85,B 0,C 180,E1 -8387.725,E2 -8387.725} C_VEL
LIN {X 0,Y 456.96,Z 443.822,A -85,B 0,C 180,E1 -8387.973,E2 -8387.973} C_VEL
LIN {X 0,Y 455.877,Z 433.115,A -85,B 0,C 180,E1 -8388.482,E2 -8388.482} C_VEL
LIN {X 0,Y 454.593,Z 417.41,A -85,B 0,C 180,E1 -8389.059,E2 -8389.059} C_VEL
LIN {X 0,Y 453.36,Z 408.134,A -85,B 0,C 180,E1 -8389.364,E2 -8389.364} C_VEL
LIN {X 0,Y 453.339,Z 407.29,A -85,B 0,C 180,E1 -8389.471,E2 -8389.471} C_VEL
LIN {X 0,Y 453.528,Z 391.465,A -85,B 0,C 180,E1 -8393.035,E2 -8393.035} C_VEL
LIN {X 0,Y 453.74,Z 377.187,A -85,B 0,C 180,E1 -8396.324,E2 -8396.324} C_VEL
LIN {X 0,Y 453.971,Z 364.087,A -85,B 0,C 180,E1 -8399.442,E2 -8399.442} C_VEL
LIN {X 0,Y 454.251,Z 350.696,A -85,B 0,C 180,E1 -8402.787,E2 -8402.787} C_VEL
LIN {X 0,Y 455.04,Z 336.628,A -85,B 0,C 180,E1 -8406.57,E2 -8406.57} C_VEL
LIN {X 0,Y 455.779,Z 329.524,A -85,B 0,C 180,E1 -8408.646,E2 -8408.646} C_VEL
LIN {X 0,Y 455.306,Z 325.7,A -85,B 0,C 180,E1 -8409.918,E2 -8409.918} C_VEL
LIN {X 0,Y 453.921,Z 318.742,A -85,B 0,C 180,E1 -8412.563,E2 -8412.563} C_VEL
LIN {X 0,Y 453.467,Z 316.67,A -85,B 0,C 180,E1 -8413.509,E2 -8413.509} C_VEL
LIN {X 0,Y 453.469,Z 316.627,A -85,B 0,C 180,E1 -8415.779,E2 -8415.779} C_VEL
LIN {X 0,Y 453.519,Z 316.621,A -85,B 0,C 180,E1 -8419.406,E2 -8419.406} C_VEL
LIN {X 0,Y 453.48,Z 316.623,A -85,B 0,C 180,E1 -8422.223,E2 -8422.223} C_VEL
LIN {X 0,Y 453.493,Z 316.624,A -85,B 0,C 180,E1 -8425.223,E2 -8425.223} C_VEL
LIN {X 0,Y 453.469,Z 316.623,A -85,B 0,C 180,E1 -8428.475,E2 -8428.475} C_VEL
LIN {X 0,Y 453.536,Z 316.616,A -85,B 0,C 180,E1 -8432.041,E2 -8432.041} C_VEL
LIN {X 0,Y 453.518,Z 316.62,A -85,B 0,C 180,E1 -8435.266,E2 -8435.266} C_VEL
LIN {X 0,Y 453.484,Z 316.625,A -85,B 0,C 180,E1 -8438.415,E2 -8438.415} C_VEL
LIN {X 0,Y 453.552,Z 316.785,A -85,B 0,C 180,E1 -8440.353,E2 -8440.353} C_VEL
LIN {X 0,Y 453.86,Z 317.999,A -85,B 0,C 180,E1 -8440.535,E2 -8440.535} C_VEL
LIN {X 0,Y 458.324,Z 330.609,A -85,B 0,C 180,E1 -8441.447,E2 -8441.447} C_VEL
LIN {X 0,Y 458.702,Z 332.53,A -85,B 0,C 180,E1 -8441.579,E2 -8441.579} C_VEL
LIN {X 0,Y 458.103,Z 345.331,A -85,B 0,C 180,E1 -8442.416,E2 -8442.416} C_VEL
LIN {X 0,Y 457.347,Z 358.291,A -85,B 0,C 180,E1 -8443.484,E2 -8443.484} C_VEL
LIN {X 0,Y 456.709,Z 369.328,A -85,B 0,C 180,E1 -8444.607,E2 -8444.607} C_VEL
LIN {X 0,Y 456.12,Z 378.497,A -85,B 0,C 180,E1 -8445.728,E2 -8445.728} C_VEL
LIN {X 0,Y 455.43,Z 387.7,A -85,B 0,C 180,E1 -8447.07,E2 -8447.07} C_VEL
LIN {X 0,Y 454.907,Z 395.29,A -85,B 0,C 180,E1 -8448.414,E2 -8448.414} C_VEL
LIN {X 0,Y 454.469,Z 401.565,A -85,B 0,C 180,E1 -8449.756,E2 -8449.756} C_VEL
LIN {X 0,Y 454.125,Z 406.745,A -85,B 0,C 180,E1 -8451.097,E2 -8451.097} C_VEL
LIN {X 0,Y 453.738,Z 412.114,A -85,B 0,C 180,E1 -8452.882,E2 -8452.882} C_VEL
LIN {X 0,Y 453.652,Z 414.201,A -85,B 0,C 180,E1 -8453.775,E2 -8453.775} C_VEL
LIN {X 0,Y 453.32,Z 417.317,A -85,B 0,C 180,E1 -8455.554,E2 -8455.554} C_VEL
LIN {X 0,Y 453.205,Z 419.04,A -85,B 0,C 180,E1 -8457.334,E2 -8457.334} C_VEL
LIN {X 0,Y 453.133,Z 419.421,A -85,B 0,C 180,E1 -8459.112,E2 -8459.112} C_VEL
LIN {X 0,Y 453.109,Z 418.468,A -85,B 0,C 180,E1 -8460.889,E2 -8460.889} C_VEL
LIN {X 0,Y 453.131,Z 416.185,A -85,B 0,C 180,E1 -8462.667,E2 -8462.667} C_VEL
LIN {X 0,Y 453.353,Z 412.5,A -85,B 0,C 180,E1 -8464.446,E2 -8464.446} C_VEL
LIN {X 0,Y 453.575,Z 407.334,A -85,B 0,C 180,E1 -8466.227,E2 -8466.227} C_VEL
LIN {X 0,Y 453.938,Z 401.584,A -85,B 0,C 180,E1 -8467.747,E2 -8467.747} C_VEL
LIN {X 0,Y 454.341,Z 394.064,A -85,B 0,C 180,E1 -8469.348,E2 -8469.348} C_VEL
LIN {X 0,Y 454.758,Z 386.365,A -85,B 0,C 180,E1 -8470.688,E2 -8470.688} C_VEL
LIN {X 0,Y 455.284,Z 377.133,A -85,B 0,C 180,E1 -8472.028,E2 -8472.028} C_VEL
LIN {X 0,Y 455.97,Z 366.941,A -85,B 0,C 180,E1 -8473.255,E2 -8473.255} C_VEL
LIN {X 0,Y 456.592,Z 355.758,A -85,B 0,C 180,E1 -8474.371,E2 -8474.371} C_VEL
LIN {X 0,Y 457.242,Z 343.47,A -85,B 0,C 180,E1 -8475.376,E2 -8475.376} C_VEL
LIN {X 0,Y 457.779,Z 331.083,A -85,B 0,C 180,E1 -8476.197,E2 -8476.197} C_VEL
LIN {X 0,Y 453.649,Z 317.152,A -85,B 0,C 180,E1 -8477.148,E2 -8477.148} C_VEL
LIN {X 0,Y 453.533,Z 316.638,A -85,B 0,C 180,E1 -8477.356,E2 -8477.356} C_VEL
LIN {X 0,Y 453.509,Z 316.62,A -85,B 0,C 180,E1 -8479.934,E2 -8479.934} C_VEL
LIN {X 0,Y 453.484,Z 316.626,A -85,B 0,C 180,E1 -8482.796,E2 -8482.796} C_VEL
LIN {X 0,Y 453.522,Z 316.613,A -85,B 0,C 180,E1 -8485.999,E2 -8485.999} C_VEL
LIN {X 0,Y 453.514,Z 316.621,A -85,B 0,C 180,E1 -8488.712,E2 -8488.712} C_VEL
LIN {X 0,Y 453.469,Z 316.62,A -85,B 0,C 180,E1 -8491.8,E2 -8491.8} C_VEL
LIN {X 0,Y 453.487,Z 316.62,A -85,B 0,C 180,E1 -8494.989,E2 -8494.989} C_VEL
LIN {X 0,Y 453.466,Z 316.625,A -85,B 0,C 180,E1 -8498.312,E2 -8498.312} C_VEL
LIN {X 0,Y 453.499,Z 316.622,A -85,B 0,C 180,E1 -8500.609,E2 -8500.609} C_VEL
LIN {X 0,Y 453.459,Z 316.621,A -85,B 0,C 180,E1 -8503.244,E2 -8503.244} C_VEL
LIN {X 0,Y 453.479,Z 316.619,A -85,B 0,C 180,E1 -8505.78,E2 -8505.78} C_VEL
LIN {X 0,Y 453.487,Z 316.623,A -85,B 0,C 180,E1 -8508.21,E2 -8508.21} C_VEL
LIN {X 0,Y 453.521,Z 316.615,A -85,B 0,C 180,E1 -8510.79,E2 -8510.79} C_VEL
LIN {X 0,Y 453.46,Z 316.624,A -85,B 0,C 180,E1 -8513.917,E2 -8513.917} C_VEL
LIN {X 0,Y 453.489,Z 316.617,A -85,B 0,C 180,E1 -8517.151,E2 -8517.151} C_VEL
LIN {X 0,Y 453.481,Z 316.625,A -85,B 0,C 180,E1 -8520.268,E2 -8520.268} C_VEL
LIN {X 0,Y 453.511,Z 316.614,A -85,B 0,C 180,E1 -8523.294,E2 -8523.294} C_VEL
LIN {X 0,Y 453.504,Z 316.621,A -85,B 0,C 180,E1 -8526.238,E2 -8526.238} C_VEL
LIN {X 0,Y 453.489,Z 316.617,A -85,B 0,C 180,E1 -8529.117,E2 -8529.117} C_VEL
LIN {X 0,Y 453.519,Z 316.62,A -85,B 0,C 180,E1 -8531.944,E2 -8531.944} C_VEL
LIN {X 0,Y 453.546,Z 316.61,A -85,B 0,C 180,E1 -8534.726,E2 -8534.726} C_VEL
LIN {X 0,Y 453.555,Z 316.61,A -85,B 0,C 180,E1 -8538.092,E2 -8538.092} C_VEL
LIN {X 0,Y 452.904,Z 316.694,A -85,B 0,C 180,E1 -8538.833,E2 -8538.833} C_VEL
LIN {X 0,Y 450.062,Z 317.056,A -85,B 0,C 180,E1 -8540.037,E2 -8540.037} C_VEL
LIN {X 0,Y 447.673,Z 317.355,A -85,B 0,C 180,E1 -8541.008,E2 -8541.008} C_VEL
LIN {X 0,Y 446.68,Z 317.474,A -85,B 0,C 180,E1 -8541.758,E2 -8541.758} C_VEL
LIN {X 0,Y 446.616,Z 317.479,A -85,B 0,C 180,E1 -8542.012,E2 -8542.012} C_VEL
LIN {X 0,Y 446.647,Z 317.47,A -85,B 0,C 180,E1 -8544.582,E2 -8544.582} C_VEL
LIN {X 0,Y 446.669,Z 317.469,A -85,B 0,C 180,E1 -8548.196,E2 -8548.196} C_VEL
LIN {X 0,Y 446.798,Z 317.455,A -85,B 0,C 180,E1 -8549.999,E2 -8549.999} C_VEL
LIN {X 0,Y 446.696,Z 317.463,A -85,B 0,C 180,E1 -8552.705,E2 -8552.705} C_VEL
LIN {X 0,Y 446.651,Z 317.47,A -85,B 0,C 180,E1 -8556.323,E2 -8556.323} C_VEL
LIN {X 0,Y 446.542,Z 317.484,A -85,B 0,C 180,E1 -8559.054,E2 -8559.054} C_VEL
LIN {X 0,Y 446.525,Z 317.485,A -85,B 0,C 180,E1 -8562.729,E2 -8562.729} C_VEL
LIN {X 0,Y 446.499,Z 317.488,A -85,B 0,C 180,E1 -8566.227,E2 -8566.227} C_VEL
LIN {X 0,Y 446.472,Z 317.497,A -85,B 0,C 180,E1 -8569.302,E2 -8569.302} C_VEL
LIN {X 0,Y 446.42,Z 317.498,A -85,B 0,C 180,E1 -8572.198,E2 -8572.198} C_VEL
LIN {X 0,Y 446.459,Z 317.498,A -85,B 0,C 180,E1 -8575.151,E2 -8575.151} C_VEL
LIN {X 0,Y 446.485,Z 317.49,A -85,B 0,C 180,E1 -8578.177,E2 -8578.177} C_VEL
LIN {X 0,Y 446.42,Z 317.499,A -85,B 0,C 180,E1 -8581.774,E2 -8581.774} C_VEL
LIN {X 0,Y 446.428,Z 317.497,A -85,B 0,C 180,E1 -8584.522,E2 -8584.522} C_VEL
LIN {X 0,Y 446.414,Z 317.498,A -85,B 0,C 180,E1 -8588.078,E2 -8588.078} C_VEL
LIN {X 0,Y 446.426,Z 317.502,A -85,B 0,C 180,E1 -8590.917,E2 -8590.917} C_VEL
LIN {X 0,Y 446.42,Z 317.498,A -85,B 0,C 180,E1 -8593.842,E2 -8593.842} C_VEL
LIN {X 0,Y 446.418,Z 317.499,A -85,B 0,C 180,E1 -8596.399,E2 -8596.399} C_VEL
LIN {X 0,Y 446.447,Z 317.494,A -85,B 0,C 180,E1 -8599.802,E2 -8599.802} C_VEL
LIN {X 0,Y 446.425,Z 317.497,A -85,B 0,C 180,E1 -8602.122,E2 -8602.122} C_VEL
LIN {X 0,Y 446.425,Z 317.498,A -85,B 0,C 180,E1 -8605.476,E2 -8605.476} C_VEL
LIN {X 0,Y 446.429,Z 317.502,A -85,B 0,C 180,E1 -8608.7,E2 -8608.7} C_VEL
LIN {X 0,Y 446.478,Z 317.49,A -85,B 0,C 180,E1 -8611.821,E2 -8611.821} C_VEL
LIN {X 0,Y 446.453,Z 317.5,A -85,B 0,C 180,E1 -8614.847,E2 -8614.847} C_VEL
LIN {X 0,Y 446.441,Z 317.497,A -85,B 0,C 180,E1 -8618.244,E2 -8618.244} C_VEL
LIN {X 0,Y 446.451,Z 317.494,A -85,B 0,C 180,E1 -8621.649,E2 -8621.649} C_VEL
LIN {X 0,Y 446.5,Z 317.494,A -85,B 0,C 180,E1 -8624.479,E2 -8624.479} C_VEL
LIN {X 0,Y 446.51,Z 317.49,A -85,B 0,C 180,E1 -8628.193,E2 -8628.193} C_VEL
LIN {X 0,Y 446.592,Z 317.477,A -85,B 0,C 180,E1 -8631.857,E2 -8631.857} C_VEL
LIN {X 0,Y 446.639,Z 317.477,A -85,B 0,C 180,E1 -8634.582,E2 -8634.582} C_VEL
LIN {X 0,Y 446.703,Z 317.462,A -85,B 0,C 180,E1 -8637.294,E2 -8637.294} C_VEL
LIN {X 0,Y 446.786,Z 317.455,A -85,B 0,C 180,E1 -8640,E2 -8640} C_VEL
LIN {X 0,Y 446.702,Z 317.466,A -85,B 0,C 180,E1 -8642.705,E2 -8642.705} C_VEL
LIN {X 0,Y 446.639,Z 317.478,A -85,B 0,C 180,E1 -8646.324,E2 -8646.324} C_VEL
LIN {X 0,Y 446.531,Z 317.484,A -85,B 0,C 180,E1 -8649.055,E2 -8649.055} C_VEL
LIN {X 0,Y 446.525,Z 317.486,A -85,B 0,C 180,E1 -8652.729,E2 -8652.729} C_VEL
LIN {X 0,Y 446.487,Z 317.493,A -85,B 0,C 180,E1 -8656.459,E2 -8656.459} C_VEL
LIN {X 0,Y 446.461,Z 317.493,A -85,B 0,C 180,E1 -8659.303,E2 -8659.303} C_VEL
LIN {X 0,Y 446.411,Z 317.504,A -85,B 0,C 180,E1 -8662.2,E2 -8662.2} C_VEL
LIN {X 0,Y 446.45,Z 317.494,A -85,B 0,C 180,E1 -8665.153,E2 -8665.153} C_VEL
LIN {X 0,Y 446.477,Z 317.495,A -85,B 0,C 180,E1 -8668.179,E2 -8668.179} C_VEL
LIN {X 0,Y 446.423,Z 317.498,A -85,B 0,C 180,E1 -8671.3,E2 -8671.3} C_VEL
LIN {X 0,Y 446.423,Z 317.498,A -85,B 0,C 180,E1 -8674.523,E2 -8674.523} C_VEL
LIN {X 0,Y 446.432,Z 317.503,A -85,B 0,C 180,E1 -8678.084,E2 -8678.084} C_VEL
LIN {X 0,Y 446.437,Z 317.5,A -85,B 0,C 180,E1 -8680.921,E2 -8680.921} C_VEL
LIN {X 0,Y 446.46,Z 317.613,A -85,B 0,C 180,E1 -8684.374,E2 -8684.374} C_VEL
LIN {X 0,Y 448.572,Z 327.681,A -85,B 0,C 180,E1 -8687.648,E2 -8687.648} C_VEL
LIN {X 0,Y 450.16,Z 335.965,A -85,B 0,C 180,E1 -8690.202,E2 -8690.202} C_VEL
LIN {X 0,Y 450.191,Z 339.988,A -85,B 0,C 180,E1 -8691.36,E2 -8691.36} C_VEL
LIN {X 0,Y 449.102,Z 353.834,A -85,B 0,C 180,E1 -8695.168,E2 -8695.168} C_VEL
LIN {X 0,Y 448.274,Z 367.613,A -85,B 0,C 180,E1 -8698.845,E2 -8698.845} C_VEL
LIN {X 0,Y 447.736,Z 377.913,A -85,B 0,C 180,E1 -8701.524,E2 -8701.524} C_VEL
LIN {X 0,Y 447.267,Z 389.16,A -85,B 0,C 180,E1 -8704.399,E2 -8704.399} C_VEL
LIN {X 0,Y 446.84,Z 400.855,A -85,B 0,C 180,E1 -8707.336,E2 -8707.336} C_VEL
LIN {X 0,Y 446.426,Z 413.844,A -85,B 0,C 180,E1 -8710.508,E2 -8710.508} C_VEL
LIN {X 0,Y 447.04,Z 418.716,A -85,B 0,C 180,E1 -8710.685,E2 -8710.685} C_VEL
LIN {X 0,Y 449.068,Z 433.801,A -85,B 0,C 180,E1 -8711.196,E2 -8711.196} C_VEL
LIN {X 0,Y 450.451,Z 446.487,A -85,B 0,C 180,E1 -8711.765,E2 -8711.765} C_VEL
LIN {X 0,Y 449.762,Z 459.769,A -85,B 0,C 180,E1 -8712.46,E2 -8712.46} C_VEL
LIN {X 0,Y 448.978,Z 472.221,A -85,B 0,C 180,E1 -8713.285,E2 -8713.285} C_VEL
LIN {X 0,Y 448.197,Z 484.681,A -85,B 0,C 180,E1 -8714.308,E2 -8714.308} C_VEL
LIN {X 0,Y 447.492,Z 496.065,A -85,B 0,C 180,E1 -8715.447,E2 -8715.447} C_VEL
LIN {X 0,Y 446.799,Z 507.288,A -85,B 0,C 180,E1 -8716.817,E2 -8716.817} C_VEL
LIN {X 0,Y 446.42,Z 516.591,A -85,B 0,C 180,E1 -8718.191,E2 -8718.191} C_VEL
LIN {X 0,Y 446.009,Z 525.48,A -85,B 0,C 180,E1 -8719.79,E2 -8719.79} C_VEL
LIN {X 0,Y 445.818,Z 532.667,A -85,B 0,C 180,E1 -8721.388,E2 -8721.388} C_VEL
LIN {X 0,Y 445.759,Z 537.647,A -85,B 0,C 180,E1 -8722.755,E2 -8722.755} C_VEL
LIN {X 0,Y 445.782,Z 541.667,A -85,B 0,C 180,E1 -8724.119,E2 -8724.119} C_VEL
LIN {X 0,Y 445.787,Z 544.705,A -85,B 0,C 180,E1 -8725.48,E2 -8725.48} C_VEL
LIN {X 0,Y 445.815,Z 547.467,A -85,B 0,C 180,E1 -8727.29,E2 -8727.29} C_VEL
LIN {X 0,Y 445.804,Z 548.759,A -85,B 0,C 180,E1 -8729.098,E2 -8729.098} C_VEL
LIN {X 0,Y 445.964,Z 548.889,A -85,B 0,C 180,E1 -8730.001,E2 -8730.001} C_VEL
LIN {X 0,Y 445.984,Z 548.634,A -85,B 0,C 180,E1 -8730.904,E2 -8730.904} C_VEL
LIN {X 0,Y 445.871,Z 547.005,A -85,B 0,C 180,E1 -8732.711,E2 -8732.711} C_VEL
LIN {X 0,Y 445.969,Z 543.913,A -85,B 0,C 180,E1 -8734.52,E2 -8734.52} C_VEL
LIN {X 0,Y 445.883,Z 539.231,A -85,B 0,C 180,E1 -8736.335,E2 -8736.335} C_VEL
LIN {X 0,Y 445.878,Z 534.643,A -85,B 0,C 180,E1 -8737.7,E2 -8737.7} C_VEL
LIN {X 0,Y 445.98,Z 527.943,A -85,B 0,C 180,E1 -8739.296,E2 -8739.296} C_VEL
LIN {X 0,Y 446.17,Z 519.626,A -85,B 0,C 180,E1 -8740.896,E2 -8740.896} C_VEL
LIN {X 0,Y 446.461,Z 509.785,A -85,B 0,C 180,E1 -8742.447,E2 -8742.447} C_VEL
LIN {X 0,Y 447.059,Z 498.827,A -85,B 0,C 180,E1 -8743.872,E2 -8743.872} C_VEL
LIN {X 0,Y 447.653,Z 487.181,A -85,B 0,C 180,E1 -8745.131,E2 -8745.131} C_VEL
LIN {X 0,Y 448.459,Z 474.367,A -85,B 0,C 180,E1 -8746.268,E2 -8746.268} C_VEL
LIN {X 0,Y 449.25,Z 461.986,A -85,B 0,C 180,E1 -8747.175,E2 -8747.175} C_VEL
LIN {X 0,Y 450.116,Z 447.407,A -85,B 0,C 180,E1 -8748.03,E2 -8748.03} C_VEL
LIN {X 0,Y 449.525,Z 439.962,A -85,B 0,C 180,E1 -8748.428,E2 -8748.428} C_VEL
LIN {X 0,Y 448.443,Z 424.401,A -85,B 0,C 180,E1 -8749.115,E2 -8749.115} C_VEL
LIN {X 0,Y 446.577,Z 408.869,A -85,B 0,C 180,E1 -8749.658,E2 -8749.658} C_VEL
LIN {X 0,Y 446.305,Z 406.334,A -85,B 0,C 180,E1 -8749.772,E2 -8749.772} C_VEL
LIN {X 0,Y 446.425,Z 392.365,A -85,B 0,C 180,E1 -8752.932,E2 -8752.932} C_VEL
LIN {X 0,Y 446.648,Z 378.259,A -85,B 0,C 180,E1 -8756.247,E2 -8756.247} C_VEL
LIN {X 0,Y 446.902,Z 366.173,A -85,B 0,C 180,E1 -8759.178,E2 -8759.178} C_VEL
LIN {X 0,Y 447.162,Z 353.854,A -85,B 0,C 180,E1 -8762.302,E2 -8762.302} C_VEL
LIN {X 0,Y 447.892,Z 340.08,A -85,B 0,C 180,E1 -8766.046,E2 -8766.046} C_VEL
LIN {X 0,Y 448.858,Z 330.873,A -85,B 0,C 180,E1 -8768.778,E2 -8768.778} C_VEL
LIN {X 0,Y 448.425,Z 327.349,A -85,B 0,C 180,E1 -8769.985,E2 -8769.985} C_VEL
LIN {X 0,Y 447.135,Z 320.814,A -85,B 0,C 180,E1 -8772.522,E2 -8772.522} C_VEL
LIN {X 0,Y 446.429,Z 317.556,A -85,B 0,C 180,E1 -8774,E2 -8774} C_VEL
LIN {X 0,Y 446.403,Z 317.507,A -85,B 0,C 180,E1 -8776.404,E2 -8776.404} C_VEL
LIN {X 0,Y 446.471,Z 317.498,A -85,B 0,C 180,E1 -8779.805,E2 -8779.805} C_VEL
LIN {X 0,Y 446.436,Z 317.501,A -85,B 0,C 180,E1 -8782.124,E2 -8782.124} C_VEL
LIN {X 0,Y 446.434,Z 317.502,A -85,B 0,C 180,E1 -8785.478,E2 -8785.478} C_VEL
LIN {X 0,Y 446.419,Z 317.501,A -85,B 0,C 180,E1 -8788.7,E2 -8788.7} C_VEL
LIN {X 0,Y 446.488,Z 317.495,A -85,B 0,C 180,E1 -8791.822,E2 -8791.822} C_VEL
LIN {X 0,Y 446.461,Z 317.499,A -85,B 0,C 180,E1 -8794.848,E2 -8794.848} C_VEL
LIN {X 0,Y 446.452,Z 317.501,A -85,B 0,C 180,E1 -8798.245,E2 -8798.245} C_VEL
LIN {X 0,Y 446.503,Z 317.699,A -85,B 0,C 180,E1 -8799.98,E2 -8799.98} C_VEL
LIN {X 0,Y 446.771,Z 318.772,A -85,B 0,C 180,E1 -8800.144,E2 -8800.144} C_VEL
LIN {X 0,Y 451.332,Z 331.264,A -85,B 0,C 180,E1 -8801.082,E2 -8801.082} C_VEL
LIN {X 0,Y 452.131,Z 334.157,A -85,B 0,C 180,E1 -8801.301,E2 -8801.301} C_VEL
LIN {X 0,Y 451.478,Z 346.602,A -85,B 0,C 180,E1 -8802.133,E2 -8802.133} C_VEL
LIN {X 0,Y 450.758,Z 358.459,A -85,B 0,C 180,E1 -8803.119,E2 -8803.119} C_VEL
LIN {X 0,Y 450.039,Z 369.629,A -85,B 0,C 180,E1 -8804.256,E2 -8804.256} C_VEL
LIN {X 0,Y 449.366,Z 379.757,A -85,B 0,C 180,E1 -8805.509,E2 -8805.509} C_VEL
LIN {X 0,Y 448.701,Z 387.526,A -85,B 0,C 180,E1 -8806.643,E2 -8806.643} C_VEL
LIN {X 0,Y 448.065,Z 396.477,A -85,B 0,C 180,E1 -8808.235,E2 -8808.235} C_VEL
LIN {X 0,Y 447.58,Z 402.739,A -85,B 0,C 180,E1 -8809.597,E2 -8809.597} C_VEL
LIN {X 0,Y 447.208,Z 407.897,A -85,B 0,C 180,E1 -8810.959,E2 -8810.959} C_VEL
LIN {X 0,Y 446.792,Z 413.238,A -85,B 0,C 180,E1 -8812.771,E2 -8812.771} C_VEL
LIN {X 0,Y 446.682,Z 415.313,A -85,B 0,C 180,E1 -8813.677,E2 -8813.677} C_VEL
LIN {X 0,Y 446.322,Z 418.415,A -85,B 0,C 180,E1 -8815.485,E2 -8815.485} C_VEL
LIN {X 0,Y 446.209,Z 420.112,A -85,B 0,C 180,E1 -8817.292,E2 -8817.292} C_VEL
LIN {X 0,Y 446.136,Z 420.464,A -85,B 0,C 180,E1 -8819.098,E2 -8819.098} C_VEL
LIN {X 0,Y 446.089,Z 419.484,A -85,B 0,C 180,E1 -8820.903,E2 -8820.903} C_VEL
LIN {X 0,Y 446.108,Z 417.169,A -85,B 0,C 180,E1 -8822.709,E2 -8822.709} C_VEL
LIN {X 0,Y 446.339,Z 413.448,A -85,B 0,C 180,E1 -8824.516,E2 -8824.516} C_VEL
LIN {X 0,Y 446.589,Z 408.241,A -85,B 0,C 180,E1 -8826.325,E2 -8826.325} C_VEL
LIN {X 0,Y 446.974,Z 402.454,A -85,B 0,C 180,E1 -8827.867,E2 -8827.867} C_VEL
LIN {X 0,Y 447.403,Z 394.89,A -85,B 0,C 180,E1 -8829.494,E2 -8829.494} C_VEL
LIN {X 0,Y 447.833,Z 387.149,A -85,B 0,C 180,E1 -8830.855,E2 -8830.855} C_VEL
LIN {X 0,Y 448.396,Z 377.871,A -85,B 0,C 180,E1 -8832.216,E2 -8832.216} C_VEL
LIN {X 0,Y 449.096,Z 367.623,A -85,B 0,C 180,E1 -8833.461,E2 -8833.461} C_VEL
LIN {X 0,Y 449.767,Z 356.373,A -85,B 0,C 180,E1 -8834.594,E2 -8834.594} C_VEL
LIN {X 0,Y 450.439,Z 344.027,A -85,B 0,C 180,E1 -8835.614,E2 -8835.614} C_VEL
LIN {X 0,Y 450.87,Z 332.069,A -85,B 0,C 180,E1 -8836.423,E2 -8836.423} C_VEL
LIN {X 0,Y 446.595,Z 318.079,A -85,B 0,C 180,E1 -8837.398,E2 -8837.398} C_VEL
LIN {X 0,Y 446.498,Z 317.525,A -85,B 0,C 180,E1 -8837.579,E2 -8837.579} C_VEL
LIN {X 0,Y 446.449,Z 317.5,A -85,B 0,C 180,E1 -8840.263,E2 -8840.263} C_VEL
LIN {X 0,Y 446.433,Z 317.501,A -85,B 0,C 180,E1 -8843.177,E2 -8843.177} C_VEL
LIN {X 0,Y 446.48,Z 317.492,A -85,B 0,C 180,E1 -8846.203,E2 -8846.203} C_VEL
LIN {X 0,Y 446.453,Z 317.495,A -85,B 0,C 180,E1 -8849.209,E2 -8849.209} C_VEL
LIN {X 0,Y 446.427,Z 317.501,A -85,B 0,C 180,E1 -8852.362,E2 -8852.362} C_VEL
LIN {X 0,Y 446.426,Z 317.497,A -85,B 0,C 180,E1 -8855.626,E2 -8855.626} C_VEL
LIN {X 0,Y 446.443,Z 317.497,A -85,B 0,C 180,E1 -8859.028,E2 -8859.028} C_VEL
LIN {X 0,Y 446.439,Z 317.501,A -85,B 0,C 180,E1 -8862.277,E2 -8862.277} C_VEL
LIN {X 0,Y 446.461,Z 317.493,A -85,B 0,C 180,E1 -8865.103,E2 -8865.103} C_VEL
LIN {X 0,Y 446.435,Z 317.5,A -85,B 0,C 180,E1 -8868.609,E2 -8868.609} C_VEL
LIN {X 0,Y 446.466,Z 317.493,A -85,B 0,C 180,E1 -8870.975,E2 -8870.975} C_VEL
LIN {X 0,Y 446.425,Z 317.504,A -85,B 0,C 180,E1 -8874.374,E2 -8874.374} C_VEL
LIN {X 0,Y 446.428,Z 317.498,A -85,B 0,C 180,E1 -8877.638,E2 -8877.638} C_VEL
LIN {X 0,Y 446.455,Z 317.494,A -85,B 0,C 180,E1 -8880.79,E2 -8880.79} C_VEL
LIN {X 0,Y 446.484,Z 317.494,A -85,B 0,C 180,E1 -8883.848,E2 -8883.848} C_VEL
LIN {X 0,Y 446.432,Z 317.497,A -85,B 0,C 180,E1 -8886.823,E2 -8886.823} C_VEL
LIN {X 0,Y 446.451,Z 317.498,A -85,B 0,C 180,E1 -8889.737,E2 -8889.737} C_VEL
LIN {X 0,Y 446.47,Z 317.493,A -85,B 0,C 180,E1 -8892.597,E2 -8892.597} C_VEL
LIN {X 0,Y 446.477,Z 317.492,A -85,B 0,C 180,E1 -8895.412,E2 -8895.412} C_VEL
LIN {X 0,Y 446.524,Z 317.489,A -85,B 0,C 180,E1 -8898.192,E2 -8898.192} C_VEL
LIN {X 0,Y 446.606,Z 317.482,A -85,B 0,C 180,E1 -8901.857,E2 -8901.857} C_VEL
LIN {X 0,Y 446.616,Z 317.479,A -85,B 0,C 180,E1 -8902.012,E2 -8902.012} C_VEL
LIN {X 0,Y 445.977,Z 317.554,A -85,B 0,C 180,E1 -8902.766,E2 -8902.766} C_VEL
LIN {X 0,Y 443.058,Z 317.922,A -85,B 0,C 180,E1 -8903.988,E2 -8903.988} C_VEL
LIN {X 0,Y 440.567,Z 318.23,A -85,B 0,C 180,E1 -8904.975,E2 -8904.975} C_VEL
LIN {X 0,Y 439.502,Z 318.366,A -85,B 0,C 180,E1 -8905.739,E2 -8905.739} C_VEL
LIN {X 0,Y 439.42,Z 318.37,A -85,B 0,C 180,E1 -8905.997,E2 -8905.997} C_VEL
LIN {X 0,Y 439.639,Z 318.345,A -85,B 0,C 180,E1 -8908.167,E2 -8908.167} C_VEL
LIN {X 0,Y 439.768,Z 318.331,A -85,B 0,C 180,E1 -8909.999,E2 -8909.999} C_VEL
LIN {X 0,Y 439.646,Z 318.341,A -85,B 0,C 180,E1 -8912.748,E2 -8912.748} C_VEL
LIN {X 0,Y 439.623,Z 318.345,A -85,B 0,C 180,E1 -8916.424,E2 -8916.424} C_VEL
LIN {X 0,Y 439.504,Z 318.362,A -85,B 0,C 180,E1 -8919.201,E2 -8919.201} C_VEL
LIN {X 0,Y 439.469,Z 318.365,A -85,B 0,C 180,E1 -8922.937,E2 -8922.937} C_VEL
LIN {X 0,Y 439.45,Z 318.366,A -85,B 0,C 180,E1 -8926.348,E2 -8926.348} C_VEL
LIN {X 0,Y 439.405,Z 318.377,A -85,B 0,C 180,E1 -8929.625,E2 -8929.625} C_VEL
LIN {X 0,Y 439.367,Z 318.376,A -85,B 0,C 180,E1 -8932.574,E2 -8932.574} C_VEL
LIN {X 0,Y 439.407,Z 318.376,A -85,B 0,C 180,E1 -8935.584,E2 -8935.584} C_VEL
LIN {X 0,Y 439.418,Z 318.371,A -85,B 0,C 180,E1 -8938.672,E2 -8938.672} C_VEL
LIN {X 0,Y 439.37,Z 318.376,A -85,B 0,C 180,E1 -8942.029,E2 -8942.029} C_VEL
LIN {X 0,Y 439.393,Z 318.379,A -85,B 0,C 180,E1 -8945.339,E2 -8945.339} C_VEL
LIN {X 0,Y 439.381,Z 318.376,A -85,B 0,C 180,E1 -8948.594,E2 -8948.594} C_VEL
LIN {X 0,Y 439.387,Z 318.38,A -85,B 0,C 180,E1 -8951.256,E2 -8951.256} C_VEL
LIN {X 0,Y 439.403,Z 318.375,A -85,B 0,C 180,E1 -8954.727,E2 -8954.727} C_VEL
LIN {X 0,Y 439.393,Z 318.373,A -85,B 0,C 180,E1 -8957.795,E2 -8957.795} C_VEL
LIN {X 0,Y 439.433,Z 318.368,A -85,B 0,C 180,E1 -8960.228,E2 -8960.228} C_VEL
LIN {X 0,Y 439.372,Z 318.376,A -85,B 0,C 180,E1 -8963.712,E2 -8963.712} C_VEL
LIN {X 0,Y 439.371,Z 318.381,A -85,B 0,C 180,E1 -8967.053,E2 -8967.053} C_VEL
LIN {X 0,Y 439.392,Z 318.375,A -85,B 0,C 180,E1 -8970.274,E2 -8970.274} C_VEL
LIN {X 0,Y 439.427,Z 318.369,A -85,B 0,C 180,E1 -8973.588,E2 -8973.588} C_VEL
LIN {X 0,Y 439.381,Z 318.378,A -85,B 0,C 180,E1 -8976.429,E2 -8976.429} C_VEL
LIN {X 0,Y 439.382,Z 318.375,A -85,B 0,C 180,E1 -8979.396,E2 -8979.396} C_VEL
LIN {X 0,Y 439.425,Z 318.372,A -85,B 0,C 180,E1 -8982.309,E2 -8982.309} C_VEL
LIN {X 0,Y 439.441,Z 318.368,A -85,B 0,C 180,E1 -8985.173,E2 -8985.173} C_VEL
LIN {X 0,Y 439.476,Z 318.364,A -85,B 0,C 180,E1 -8988.001,E2 -8988.001} C_VEL
LIN {X 0,Y 439.54,Z 318.355,A -85,B 0,C 180,E1 -8991.726,E2 -8991.726} C_VEL
LIN {X 0,Y 439.614,Z 318.353,A -85,B 0,C 180,E1 -8994.495,E2 -8994.495} C_VEL
LIN {X 0,Y 439.629,Z 318.348,A -85,B 0,C 180,E1 -8998.168,E2 -8998.168} C_VEL
LIN {X 0,Y 439.756,Z 318.331,A -85,B 0,C 180,E1 -9000,E2 -9000} C_VEL
LIN {X 0,Y 439.649,Z 318.344,A -85,B 0,C 180,E1 -9002.749,E2 -9002.749} C_VEL
LIN {X 0,Y 439.61,Z 318.352,A -85,B 0,C 180,E1 -9006.425,E2 -9006.425} C_VEL
LIN {X 0,Y 439.493,Z 318.36,A -85,B 0,C 180,E1 -9009.202,E2 -9009.202} C_VEL
LIN {X 0,Y 439.496,Z 318.362,A -85,B 0,C 180,E1 -9012.727,E2 -9012.727} C_VEL
LIN {X 0,Y 439.452,Z 318.37,A -85,B 0,C 180,E1 -9016.355,E2 -9016.355} C_VEL
LIN {X 0,Y 439.394,Z 318.375,A -85,B 0,C 180,E1 -9019.626,E2 -9019.626} C_VEL
LIN {X 0,Y 439.358,Z 318.379,A -85,B 0,C 180,E1 -9022.576,E2 -9022.576} C_VEL
LIN {X 0,Y 439.397,Z 318.375,A -85,B 0,C 180,E1 -9025.585,E2 -9025.585} C_VEL
LIN {X 0,Y 439.417,Z 318.37,A -85,B 0,C 180,E1 -9028.673,E2 -9028.673} C_VEL
LIN {X 0,Y 439.376,Z 318.381,A -85,B 0,C 180,E1 -9032.034,E2 -9032.034} C_VEL
LIN {X 0,Y 439.389,Z 318.375,A -85,B 0,C 180,E1 -9035.341,E2 -9035.341} C_VEL
LIN {X 0,Y 439.393,Z 318.377,A -85,B 0,C 180,E1 -9038.594,E2 -9038.594} C_VEL
LIN {X 0,Y 439.392,Z 318.379,A -85,B 0,C 180,E1 -9041.259,E2 -9041.259} C_VEL
LIN {X 0,Y 439.434,Z 318.636,A -85,B 0,C 180,E1 -9044.089,E2 -9044.089} C_VEL
LIN {X 0,Y 441.678,Z 329.298,A -85,B 0,C 180,E1 -9047.6,E2 -9047.6} C_VEL
LIN {X 0,Y 443.234,Z 337.4,A -85,B 0,C 180,E1 -9050.141,E2 -9050.141} C_VEL
LIN {X 0,Y 443.222,Z 341.663,A -85,B 0,C 180,E1 -9051.382,E2 -9051.382} C_VEL
LIN {X 0,Y 442.13,Z 354.947,A -85,B 0,C 180,E1 -9055.094,E2 -9055.094} C_VEL
LIN {X 0,Y 441.258,Z 368.72,A -85,B 0,C 180,E1 -9058.828,E2 -9058.828} C_VEL
LIN {X 0,Y 440.648,Z 380.478,A -85,B 0,C 180,E1 -9061.934,E2 -9061.934} C_VEL
LIN {X 0,Y 440.025,Z 394.485,A -85,B 0,C 180,E1 -9065.56,E2 -9065.56} C_VEL
LIN {X 0,Y 439.517,Z 407.654,A -85,B 0,C 180,E1 -9068.914,E2 -9068.914} C_VEL
LIN {X 0,Y 439.37,Z 413.045,A -85,B 0,C 180,E1 -9070.221,E2 -9070.221} C_VEL
LIN {X 0,Y 439.918,Z 417.31,A -85,B 0,C 180,E1 -9070.38,E2 -9070.38} C_VEL
LIN {X 0,Y 442.017,Z 432.785,A -85,B 0,C 180,E1 -9070.915,E2 -9070.915} C_VEL
LIN {X 0,Y 443.503,Z 447.259,A -85,B 0,C 180,E1 -9071.585,E2 -9071.585} C_VEL
LIN {X 0,Y 442.796,Z 460.219,A -85,B 0,C 180,E1 -9072.295,E2 -9072.295} C_VEL
LIN {X 0,Y 441.983,Z 472.374,A -85,B 0,C 180,E1 -9073.131,E2 -9073.131} C_VEL
LIN {X 0,Y 441.189,Z 484.639,A -85,B 0,C 180,E1 -9074.17,E2 -9074.17} C_VEL
LIN {X 0,Y 440.467,Z 495.856,A -85,B 0,C 180,E1 -9075.328,E2 -9075.328} C_VEL
LIN {X 0,Y 439.797,Z 506.108,A -85,B 0,C 180,E1 -9076.603,E2 -9076.603} C_VEL
LIN {X 0,Y 439.378,Z 515.453,A -85,B 0,C 180,E1 -9077.999,E2 -9077.999} C_VEL
LIN {X 0,Y 438.971,Z 524.381,A -85,B 0,C 180,E1 -9079.625,E2 -9079.625} C_VEL
LIN {X 0,Y 438.764,Z 531.598,A -85,B 0,C 180,E1 -9081.248,E2 -9081.248} C_VEL
LIN {X 0,Y 438.696,Z 537.655,A -85,B 0,C 180,E1 -9082.973,E2 -9082.973} C_VEL
LIN {X 0,Y 438.712,Z 541.725,A -85,B 0,C 180,E1 -9084.485,E2 -9084.485} C_VEL
LIN {X 0,Y 438.775,Z 545.255,A -85,B 0,C 180,E1 -9086.327,E2 -9086.327} C_VEL
LIN {X 0,Y 438.773,Z 547.278,A -85,B 0,C 180,E1 -9088.165,E2 -9088.165} C_VEL
LIN {X 0,Y 438.944,Z 547.87,A -85,B 0,C 180,E1 -9090.001,E2 -9090.001} C_VEL
LIN {X 0,Y 438.965,Z 547.612,A -85,B 0,C 180,E1 -9090.918,E2 -9090.918} C_VEL
LIN {X 0,Y 438.834,Z 545.97,A -85,B 0,C 180,E1 -9092.755,E2 -9092.755} C_VEL
LIN {X 0,Y 438.908,Z 542.858,A -85,B 0,C 180,E1 -9094.593,E2 -9094.593} C_VEL
LIN {X 0,Y 438.834,Z 538.148,A -85,B 0,C 180,E1 -9096.438,E2 -9096.438} C_VEL
LIN {X 0,Y 438.836,Z 531.756,A -85,B 0,C 180,E1 -9098.288,E2 -9098.288} C_VEL
LIN {X 0,Y 438.905,Z 524.599,A -85,B 0,C 180,E1 -9099.913,E2 -9099.913} C_VEL
LIN {X 0,Y 439.163,Z 517.151,A -85,B 0,C 180,E1 -9101.306,E2 -9101.306} C_VEL
LIN {X 0,Y 439.522,Z 508.045,A -85,B 0,C 180,E1 -9102.736,E2 -9102.736} C_VEL
LIN {X 0,Y 440.031,Z 497.685,A -85,B 0,C 180,E1 -9104.098,E2 -9104.098} C_VEL
LIN {X 0,Y 440.74,Z 486.087,A -85,B 0,C 180,E1 -9105.374,E2 -9105.374} C_VEL
LIN {X 0,Y 441.555,Z 473.358,A -85,B 0,C 180,E1 -9106.53,E2 -9106.53} C_VEL
LIN {X 0,Y 442.413,Z 461.095,A -85,B 0,C 180,E1 -9107.449,E2 -9107.449} C_VEL
LIN {X 0,Y 443.295,Z 446.892,A -85,B 0,C 180,E1 -9108.307,E2 -9108.307} C_VEL
LIN {X 0,Y 442.291,Z 433.878,A -85,B 0,C 180,E1 -9109.004,E2 -9109.004} C_VEL
LIN {X 0,Y 441.083,Z 418.398,A -85,B 0,C 180,E1 -9109.658,E2 -9109.658} C_VEL
LIN {X 0,Y 439.231,Z 405.042,A -85,B 0,C 180,E1 -9110.157,E2 -9110.157} C_VEL
LIN {X 0,Y 439.214,Z 403.856,A -85,B 0,C 180,E1 -9110.343,E2 -9110.343} C_VEL
LIN {X 0,Y 439.418,Z 388.688,A -85,B 0,C 180,E1 -9113.919,E2 -9113.919} C_VEL
LIN {X 0,Y 439.676,Z 374.48,A -85,B 0,C 180,E1 -9117.359,E2 -9117.359} C_VEL
LIN {X 0,Y 439.92,Z 363.807,A -85,B 0,C 180,E1 -9120.038,E2 -9120.038} C_VEL
LIN {X 0,Y 440.246,Z 353.009,A -85,B 0,C 180,E1 -9122.873,E2 -9122.873} C_VEL
LIN {X 0,Y 441.163,Z 339.492,A -85,B 0,C 180,E1 -9126.681,E2 -9126.681} C_VEL
LIN {X 0,Y 441.939,Z 332.561,A -85,B 0,C 180,E1 -9128.81,E2 -9128.81} C_VEL
LIN {X 0,Y 441.476,Z 328.682,A -85,B 0,C 180,E1 -9130.171,E2 -9130.171} C_VEL
LIN {X 0,Y 440.225,Z 322.261,A -85,B 0,C 180,E1 -9132.746,E2 -9132.746} C_VEL
LIN {X 0,Y 439.42,Z 318.413,A -85,B 0,C 180,E1 -9134.597,E2 -9134.597} C_VEL
LIN {X 0,Y 439.4,Z 318.379,A -85,B 0,C 180,E1 -9137.796,E2 -9137.796} C_VEL
LIN {X 0,Y 439.454,Z 318.371,A -85,B 0,C 180,E1 -9140.23,E2 -9140.23} C_VEL
LIN {X 0,Y 439.381,Z 318.382,A -85,B 0,C 180,E1 -9143.714,E2 -9143.714} C_VEL
LIN {X 0,Y 439.376,Z 318.381,A -85,B 0,C 180,E1 -9147.054,E2 -9147.054} C_VEL
LIN {X 0,Y 439.385,Z 318.377,A -85,B 0,C 180,E1 -9150.275,E2 -9150.275} C_VEL
LIN {X 0,Y 439.432,Z 318.375,A -85,B 0,C 180,E1 -9153.397,E2 -9153.397} C_VEL
LIN {X 0,Y 439.39,Z 318.379,A -85,B 0,C 180,E1 -9156.43,E2 -9156.43} C_VEL
LIN {X 0,Y 439.428,Z 318.573,A -85,B 0,C 180,E1 -9159.552,E2 -9159.552} C_VEL
LIN {X 0,Y 439.778,Z 319.927,A -85,B 0,C 180,E1 -9159.748,E2 -9159.748} C_VEL
LIN {X 0,Y 443.946,Z 330.548,A -85,B 0,C 180,E1 -9160.583,E2 -9160.583} C_VEL
LIN {X 0,Y 445.577,Z 336.141,A -85,B 0,C 180,E1 -9161.029,E2 -9161.029} C_VEL
LIN {X 0,Y 444.804,Z 349.33,A -85,B 0,C 180,E1 -9161.95,E2 -9161.95} C_VEL
LIN {X 0,Y 444.05,Z 361.129,A -85,B 0,C 180,E1 -9162.975,E2 -9162.975} C_VEL
LIN {X 0,Y 443.305,Z 372.005,A -85,B 0,C 180,E1 -9164.129,E2 -9164.129} C_VEL
LIN {X 0,Y 442.644,Z 381.082,A -85,B 0,C 180,E1 -9165.284,E2 -9165.284} C_VEL
LIN {X 0,Y 441.92,Z 388.808,A -85,B 0,C 180,E1 -9166.434,E2 -9166.434} C_VEL
LIN {X 0,Y 441.327,Z 396.557,A -85,B 0,C 180,E1 -9167.819,E2 -9167.819} C_VEL
LIN {X 0,Y 440.708,Z 403.949,A -85,B 0,C 180,E1 -9169.433,E2 -9169.433} C_VEL
LIN {X 0,Y 440.312,Z 409.076,A -85,B 0,C 180,E1 -9170.816,E2 -9170.816} C_VEL
LIN {X 0,Y 439.844,Z 414.386,A -85,B 0,C 180,E1 -9172.656,E2 -9172.656} C_VEL
LIN {X 0,Y 439.711,Z 416.455,A -85,B 0,C 180,E1 -9173.576,E2 -9173.576} C_VEL
LIN {X 0,Y 439.327,Z 419.529,A -85,B 0,C 180,E1 -9175.412,E2 -9175.412} C_VEL
LIN {X 0,Y 439.21,Z 421.193,A -85,B 0,C 180,E1 -9177.249,E2 -9177.249} C_VEL
LIN {X 0,Y 439.136,Z 421.512,A -85,B 0,C 180,E1 -9179.083,E2 -9179.083} C_VEL
LIN {X 0,Y 439.068,Z 420.502,A -85,B 0,C 180,E1 -9180.917,E2 -9180.917} C_VEL
LIN {X 0,Y 439.149,Z 419.484,A -85,B 0,C 180,E1 -9181.834,E2 -9181.834} C_VEL
LIN {X 0,Y 439.187,Z 416.45,A -85,B 0,C 180,E1 -9183.67,E2 -9183.67} C_VEL
LIN {X 0,Y 439.448,Z 411.957,A -85,B 0,C 180,E1 -9185.507,E2 -9185.507} C_VEL
LIN {X 0,Y 439.886,Z 405.879,A -85,B 0,C 180,E1 -9187.344,E2 -9187.344} C_VEL
LIN {X 0,Y 440.236,Z 399.084,A -85,B 0,C 180,E1 -9188.955,E2 -9188.955} C_VEL
LIN {X 0,Y 440.811,Z 390.623,A -85,B 0,C 180,E1 -9190.565,E2 -9190.565} C_VEL
LIN {X 0,Y 441.323,Z 381.83,A -85,B 0,C 180,E1 -9191.948,E2 -9191.948} C_VEL
LIN {X 0,Y 441.923,Z 373.145,A -85,B 0,C 180,E1 -9193.099,E2 -9193.099} C_VEL
LIN {X 0,Y 442.618,Z 362.341,A -85,B 0,C 180,E1 -9194.298,E2 -9194.298} C_VEL
LIN {X 0,Y 443.24,Z 350.319,A -85,B 0,C 180,E1 -9195.402,E2 -9195.402} C_VEL
LIN {X 0,Y 443.95,Z 338.002,A -85,B 0,C 180,E1 -9196.32,E2 -9196.32} C_VEL
LIN {X 0,Y 443.92,Z 333.417,A -85,B 0,C 180,E1 -9196.627,E2 -9196.627} C_VEL
LIN {X 0,Y 439.593,Z 319.031,A -85,B 0,C 180,E1 -9197.65,E2 -9197.65} C_VEL
LIN {X 0,Y 439.477,Z 318.416,A -85,B 0,C 180,E1 -9197.809,E2 -9197.809} C_VEL
LIN {X 0,Y 439.393,Z 318.38,A -85,B 0,C 180,E1 -9200.603,E2 -9200.603} C_VEL
LIN {X 0,Y 439.42,Z 318.374,A -85,B 0,C 180,E1 -9204.265,E2 -9204.265} C_VEL
LIN {X 0,Y 439.446,Z 318.366,A -85,B 0,C 180,E1 -9207.633,E2 -9207.633} C_VEL
LIN {X 0,Y 439.366,Z 318.382,A -85,B 0,C 180,E1 -9210.789,E2 -9210.789} C_VEL
LIN {X 0,Y 439.393,Z 318.375,A -85,B 0,C 180,E1 -9214.044,E2 -9214.044} C_VEL
LIN {X 0,Y 439.354,Z 318.381,A -85,B 0,C 180,E1 -9216.887,E2 -9216.887} C_VEL
LIN {X 0,Y 439.407,Z 318.372,A -85,B 0,C 180,E1 -9219.849,E2 -9219.849} C_VEL
LIN {X 0,Y 439.386,Z 318.379,A -85,B 0,C 180,E1 -9222.627,E2 -9222.627} C_VEL
LIN {X 0,Y 439.411,Z 318.371,A -85,B 0,C 180,E1 -9225.271,E2 -9225.271} C_VEL
LIN {X 0,Y 439.395,Z 318.376,A -85,B 0,C 180,E1 -9228.743,E2 -9228.743} C_VEL
LIN {X 0,Y 439.391,Z 318.374,A -85,B 0,C 180,E1 -9231.606,E2 -9231.606} C_VEL
LIN {X 0,Y 439.405,Z 318.373,A -85,B 0,C 180,E1 -9234.844,E2 -9234.844} C_VEL
LIN {X 0,Y 439.379,Z 318.381,A -85,B 0,C 180,E1 -9238.139,E2 -9238.139} C_VEL
LIN {X 0,Y 439.439,Z 318.369,A -85,B 0,C 180,E1 -9241.598,E2 -9241.598} C_VEL
LIN {X 0,Y 439.404,Z 318.376,A -85,B 0,C 180,E1 -9244.414,E2 -9244.414} C_VEL
LIN {X 0,Y 439.37,Z 318.377,A -85,B 0,C 180,E1 -9247.424,E2 -9247.424} C_VEL
LIN {X 0,Y 439.448,Z 318.367,A -85,B 0,C 180,E1 -9250.662,E2 -9250.662} C_VEL
LIN {X 0,Y 439.469,Z 318.368,A -85,B 0,C 180,E1 -9254.224,E2 -9254.224} C_VEL
LIN {X 0,Y 439.49,Z 318.368,A -85,B 0,C 180,E1 -9258.001,E2 -9258.001} C_VEL
LIN {X 0,Y 439.554,Z 318.359,A -85,B 0,C 180,E1 -9261.726,E2 -9261.726} C_VEL
LIN {X 0,Y 439.623,Z 318.345,A -85,B 0,C 180,E1 -9264.495,E2 -9264.495} C_VEL
LIN {X 0,Y 439.42,Z 318.37,A -85,B 0,C 180,E1 -9265.997,E2 -9265.997} C_VEL
LIN {X 0,Y 438.827,Z 318.446,A -85,B 0,C 180,E1 -9266.762,E2 -9266.762} C_VEL
LIN {X 0,Y 436.204,Z 318.779,A -85,B 0,C 180,E1 -9268.01,E2 -9268.01} C_VEL
LIN {X 0,Y 433.11,Z 319.164,A -85,B 0,C 180,E1 -9269.53,E2 -9269.53} C_VEL
LIN {X 0,Y 432.725,Z 319.207,A -85,B 0,C 180,E1 -9270.052,E2 -9270.052} C_VEL
LIN {X 0,Y 432.597,Z 319.22,A -85,B 0,C 180,E1 -9272.793,E2 -9272.793} C_VEL
LIN {X 0,Y 432.577,Z 319.222,A -85,B 0,C 180,E1 -9276.529,E2 -9276.529} C_VEL
LIN {X 0,Y 432.447,Z 319.243,A -85,B 0,C 180,E1 -9279.352,E2 -9279.352} C_VEL
LIN {X 0,Y 432.434,Z 319.24,A -85,B 0,C 180,E1 -9282.802,E2 -9282.802} C_VEL
LIN {X 0,Y 432.415,Z 319.242,A -85,B 0,C 180,E1 -9286.478,E2 -9286.478} C_VEL
LIN {X 0,Y 432.341,Z 319.253,A -85,B 0,C 180,E1 -9289.959,E2 -9289.959} C_VEL
LIN {X 0,Y 432.321,Z 319.256,A -85,B 0,C 180,E1 -9292.963,E2 -9292.963} C_VEL
LIN {X 0,Y 432.365,Z 319.249,A -85,B 0,C 180,E1 -9296.031,E2 -9296.031} C_VEL
LIN {X 0,Y 432.343,Z 319.257,A -85,B 0,C 180,E1 -9299.186,E2 -9299.186} C_VEL
LIN {X 0,Y 432.323,Z 319.254,A -85,B 0,C 180,E1 -9302.442,E2 -9302.442} C_VEL
LIN {X 0,Y 432.343,Z 319.254,A -85,B 0,C 180,E1 -9305.631,E2 -9305.631} C_VEL
LIN {X 0,Y 432.348,Z 319.256,A -85,B 0,C 180,E1 -9309.342,E2 -9309.342} C_VEL
LIN {X 0,Y 432.332,Z 319.253,A -85,B 0,C 180,E1 -9311.796,E2 -9311.796} C_VEL
LIN {X 0,Y 432.338,Z 319.252,A -85,B 0,C 180,E1 -9314.345,E2 -9314.345} C_VEL
LIN {X 0,Y 432.321,Z 319.262,A -85,B 0,C 180,E1 -9317.014,E2 -9317.014} C_VEL
LIN {X 0,Y 432.337,Z 319.252,A -85,B 0,C 180,E1 -9319.818,E2 -9319.818} C_VEL
LIN {X 0,Y 432.312,Z 319.262,A -85,B 0,C 180,E1 -9323.022,E2 -9323.022} C_VEL
LIN {X 0,Y 432.354,Z 319.25,A -85,B 0,C 180,E1 -9325.995,E2 -9325.995} C_VEL
LIN {X 0,Y 432.391,Z 319.245,A -85,B 0,C 180,E1 -9329.743,E2 -9329.743} C_VEL
LIN {X 0,Y 432.394,Z 319.246,A -85,B 0,C 180,E1 -9333.371,E2 -9333.371} C_VEL
LIN {X 0,Y 432.365,Z 319.249,A -85,B 0,C 180,E1 -9336.023,E2 -9336.023} C_VEL
LIN {X 0,Y 432.343,Z 319.254,A -85,B 0,C 180,E1 -9339.045,E2 -9339.045} C_VEL
LIN {X 0,Y 432.371,Z 319.249,A -85,B 0,C 180,E1 -9342.011,E2 -9342.011} C_VEL
LIN {X 0,Y 432.389,Z 319.249,A -85,B 0,C 180,E1 -9344.926,E2 -9344.926} C_VEL
LIN {X 0,Y 432.451,Z 319.238,A -85,B 0,C 180,E1 -9347.803,E2 -9347.803} C_VEL
LIN {X 0,Y 432.484,Z 319.234,A -85,B 0,C 180,E1 -9351.59,E2 -9351.59} C_VEL
LIN {X 0,Y 432.591,Z 319.227,A -85,B 0,C 180,E1 -9354.406,E2 -9354.406} C_VEL
LIN {X 0,Y 432.598,Z 319.224,A -85,B 0,C 180,E1 -9358.138,E2 -9358.138} C_VEL
LIN {X 0,Y 432.725,Z 319.207,A -85,B 0,C 180,E1 -9360,E2 -9360} C_VEL
LIN {X 0,Y 432.598,Z 319.222,A -85,B 0,C 180,E1 -9362.793,E2 -9362.793} C_VEL
LIN {X 0,Y 432.565,Z 319.228,A -85,B 0,C 180,E1 -9366.53,E2 -9366.53} C_VEL
LIN {X 0,Y 432.436,Z 319.24,A -85,B 0,C 180,E1 -9369.353,E2 -9369.353} C_VEL
LIN {X 0,Y 432.436,Z 319.241,A -85,B 0,C 180,E1 -9372.812,E2 -9372.812} C_VEL
LIN {X 0,Y 432.415,Z 319.246,A -85,B 0,C 180,E1 -9376.484,E2 -9376.484} C_VEL
LIN {X 0,Y 432.331,Z 319.259,A -85,B 0,C 180,E1 -9379.961,E2 -9379.961} C_VEL
LIN {X 0,Y 432.312,Z 319.255,A -85,B 0,C 180,E1 -9382.964,E2 -9382.964} C_VEL
LIN {X 0,Y 432.357,Z 319.257,A -85,B 0,C 180,E1 -9386.033,E2 -9386.033} C_VEL
LIN {X 0,Y 432.345,Z 319.251,A -85,B 0,C 180,E1 -9389.187,E2 -9389.187} C_VEL
LIN {X 0,Y 432.325,Z 319.256,A -85,B 0,C 180,E1 -9392.295,E2 -9392.295} C_VEL
LIN {X 0,Y 432.334,Z 319.253,A -85,B 0,C 180,E1 -9394.677,E2 -9394.677} C_VEL
LIN {X 0,Y 432.347,Z 319.257,A -85,B 0,C 180,E1 -9398.149,E2 -9398.149} C_VEL
LIN {X 0,Y 432.36,Z 319.256,A -85,B 0,C 180,E1 -9401.608,E2 -9401.608} C_VEL
LIN {X 0,Y 432.343,Z 319.406,A -85,B 0,C 180,E1 -9403.698,E2 -9403.698} C_VEL
LIN {X 0,Y 434.541,Z 329.839,A -85,B 0,C 180,E1 -9407.214,E2 -9407.214} C_VEL
LIN {X 0,Y 436.167,Z 338.166,A -85,B 0,C 180,E1 -9409.871,E2 -9409.871} C_VEL
LIN {X 0,Y 436.316,Z 342.212,A -85,B 0,C 180,E1 -9411.084,E2 -9411.084} C_VEL
LIN {X 0,Y 435.293,Z 354.075,A -85,B 0,C 180,E1 -9414.464,E2 -9414.464} C_VEL
LIN {X 0,Y 434.35,Z 367.823,A -85,B 0,C 180,E1 -9418.275,E2 -9418.275} C_VEL
LIN {X 0,Y 433.752,Z 378.063,A -85,B 0,C 180,E1 -9421.039,E2 -9421.039} C_VEL
LIN {X 0,Y 433.191,Z 389.294,A -85,B 0,C 180,E1 -9424.022,E2 -9424.022} C_VEL
LIN {X 0,Y 432.716,Z 400.945,A -85,B 0,C 180,E1 -9427.059,E2 -9427.059} C_VEL
LIN {X 0,Y 432.293,Z 412.159,A -85,B 0,C 180,E1 -9429.915,E2 -9429.915} C_VEL
LIN {X 0,Y 432.479,Z 414.023,A -85,B 0,C 180,E1 -9430.019,E2 -9430.019} C_VEL
LIN {X 0,Y 434.659,Z 429.468,A -85,B 0,C 180,E1 -9430.536,E2 -9430.536} C_VEL
LIN {X 0,Y 436.193,Z 444.174,A -85,B 0,C 180,E1 -9431.202,E2 -9431.202} C_VEL
LIN {X 0,Y 436.571,Z 447.976,A -85,B 0,C 180,E1 -9431.402,E2 -9431.402} C_VEL
LIN {X 0,Y 435.8,Z 461.099,A -85,B 0,C 180,E1 -9432.158,E2 -9432.158} C_VEL
LIN {X 0,Y 434.945,Z 473.913,A -85,B 0,C 180,E1 -9433.092,E2 -9433.092} C_VEL
LIN {X 0,Y 433.976,Z 486.852,A -85,B 0,C 180,E1 -9434.262,E2 -9434.262} C_VEL
LIN {X 0,Y 433.244,Z 497.534,A -85,B 0,C 180,E1 -9435.438,E2 -9435.438} C_VEL
LIN {X 0,Y 432.605,Z 508.2,A -85,B 0,C 180,E1 -9436.855,E2 -9436.855} C_VEL
LIN {X 0,Y 432.172,Z 517.036,A -85,B 0,C 180,E1 -9438.272,E2 -9438.272} C_VEL
LIN {X 0,Y 431.787,Z 525.509,A -85,B 0,C 180,E1 -9439.924,E2 -9439.924} C_VEL
LIN {X 0,Y 431.677,Z 532.313,A -85,B 0,C 180,E1 -9441.575,E2 -9441.575} C_VEL
LIN {X 0,Y 431.697,Z 538.316,A -85,B 0,C 180,E1 -9443.457,E2 -9443.457} C_VEL
LIN {X 0,Y 431.693,Z 542.637,A -85,B 0,C 180,E1 -9445.332,E2 -9445.332} C_VEL
LIN {X 0,Y 431.734,Z 544.218,A -85,B 0,C 180,E1 -9446.267,E2 -9446.267} C_VEL
LIN {X 0,Y 431.742,Z 546.248,A -85,B 0,C 180,E1 -9448.135,E2 -9448.135} C_VEL
LIN {X 0,Y 431.924,Z 546.844,A -85,B 0,C 180,E1 -9450.001,E2 -9450.001} C_VEL
LIN {X 0,Y 431.945,Z 546.585,A -85,B 0,C 180,E1 -9450.933,E2 -9450.933} C_VEL
LIN {X 0,Y 431.796,Z 544.935,A -85,B 0,C 180,E1 -9452.8,E2 -9452.8} C_VEL
LIN {X 0,Y 431.852,Z 541.807,A -85,B 0,C 180,E1 -9454.668,E2 -9454.668} C_VEL
LIN {X 0,Y 431.777,Z 537.082,A -85,B 0,C 180,E1 -9456.543,E2 -9456.543} C_VEL
LIN {X 0,Y 431.762,Z 530.663,A -85,B 0,C 180,E1 -9458.425,E2 -9458.425} C_VEL
LIN {X 0,Y 431.854,Z 523.502,A -85,B 0,C 180,E1 -9460.076,E2 -9460.076} C_VEL
LIN {X 0,Y 432.157,Z 514.696,A -85,B 0,C 180,E1 -9461.73,E2 -9461.73} C_VEL
LIN {X 0,Y 432.561,Z 505.576,A -85,B 0,C 180,E1 -9463.149,E2 -9463.149} C_VEL
LIN {X 0,Y 433.171,Z 494.689,A -85,B 0,C 180,E1 -9464.566,E2 -9464.566} C_VEL
LIN {X 0,Y 433.972,Z 482.707,A -85,B 0,C 180,E1 -9465.861,E2 -9465.861} C_VEL
LIN {X 0,Y 434.8,Z 469.616,A -85,B 0,C 180,E1 -9467.03,E2 -9467.03} C_VEL
LIN {X 0,Y 435.894,Z 455.446,A -85,B 0,C 180,E1 -9468.058,E2 -9468.058} C_VEL
LIN {X 0,Y 436.36,Z 446.358,A -85,B 0,C 180,E1 -9468.609,E2 -9468.609} C_VEL
LIN {X 0,Y 435.518,Z 434.443,A -85,B 0,C 180,E1 -9469.281,E2 -9469.281} C_VEL
LIN {X 0,Y 434.364,Z 418.786,A -85,B 0,C 180,E1 -9469.986,E2 -9469.986} C_VEL
LIN {X 0,Y 432.515,Z 405.946,A -85,B 0,C 180,E1 -9470.485,E2 -9470.485} C_VEL
LIN {X 0,Y 432.122,Z 403.172,A -85,B 0,C 180,E1 -9470.624,E2 -9470.624} C_VEL
LIN {X 0,Y 432.33,Z 390.053,A -85,B 0,C 180,E1 -9473.725,E2 -9473.725} C_VEL
LIN {X 0,Y 432.594,Z 376.552,A -85,B 0,C 180,E1 -9477.059,E2 -9477.059} C_VEL
LIN {X 0,Y 432.91,Z 365.242,A -85,B 0,C 180,E1 -9479.948,E2 -9479.948} C_VEL
LIN {X 0,Y 433.264,Z 354.178,A -85,B 0,C 180,E1 -9482.917,E2 -9482.917} C_VEL
LIN {X 0,Y 434.232,Z 340.776,A -85,B 0,C 180,E1 -9486.788,E2 -9486.788} C_VEL
LIN {X 0,Y 435.035,Z 333.611,A -85,B 0,C 180,E1 -9489.054,E2 -9489.054} C_VEL
LIN {X 0,Y 434.212,Z 328.419,A -85,B 0,C 180,E1 -9490.992,E2 -9490.992} C_VEL
LIN {X 0,Y 432.925,Z 322.071,A -85,B 0,C 180,E1 -9493.748,E2 -9493.748} C_VEL
LIN {X 0,Y 432.376,Z 319.3,A -85,B 0,C 180,E1 -9495.168,E2 -9495.168} C_VEL
LIN {X 0,Y 432.37,Z 319.254,A -85,B 0,C 180,E1 -9498.393,E2 -9498.393} C_VEL
LIN {X 0,Y 432.356,Z 319.255,A -85,B 0,C 180,E1 -9501.852,E2 -9501.852} C_VEL
LIN {X 0,Y 432.344,Z 319.258,A -85,B 0,C 180,E1 -9505.323,E2 -9505.323} C_VEL
LIN {X 0,Y 432.324,Z 319.257,A -85,B 0,C 180,E1 -9508.654,E2 -9508.654} C_VEL
LIN {X 0,Y 432.385,Z 319.252,A -85,B 0,C 180,E1 -9511.877,E2 -9511.877} C_VEL
LIN {X 0,Y 432.355,Z 319.256,A -85,B 0,C 180,E1 -9514.999,E2 -9514.999} C_VEL
LIN {X 0,Y 432.361,Z 319.256,A -85,B 0,C 180,E1 -9518.046,E2 -9518.046} C_VEL
LIN {X 0,Y 432.381,Z 319.384,A -85,B 0,C 180,E1 -9519.093,E2 -9519.093} C_VEL
LIN {X 0,Y 432.674,Z 320.67,A -85,B 0,C 180,E1 -9519.297,E2 -9519.297} C_VEL
LIN {X 0,Y 437.028,Z 331.425,A -85,B 0,C 180,E1 -9520.182,E2 -9520.182} C_VEL
LIN {X 0,Y 439.04,Z 338.401,A -85,B 0,C 180,E1 -9520.76,E2 -9520.76} C_VEL
LIN {X 0,Y 438.238,Z 350.872,A -85,B 0,C 180,E1 -9521.656,E2 -9521.656} C_VEL
LIN {X 0,Y 437.443,Z 362.691,A -85,B 0,C 180,E1 -9522.709,E2 -9522.709} C_VEL
LIN {X 0,Y 436.646,Z 373.46,A -85,B 0,C 180,E1 -9523.88,E2 -9523.88} C_VEL
LIN {X 0,Y 435.927,Z 382.475,A -85,B 0,C 180,E1 -9525.052,E2 -9525.052} C_VEL
LIN {X 0,Y 435.155,Z 390.145,A -85,B 0,C 180,E1 -9526.219,E2 -9526.219} C_VEL
LIN {X 0,Y 434.43,Z 398.995,A -85,B 0,C 180,E1 -9527.86,E2 -9527.86} C_VEL
LIN {X 0,Y 433.856,Z 405.194,A -85,B 0,C 180,E1 -9529.264,E2 -9529.264} C_VEL
LIN {X 0,Y 433.404,Z 410.287,A -85,B 0,C 180,E1 -9530.668,E2 -9530.668} C_VEL
LIN {X 0,Y 432.923,Z 415.564,A -85,B 0,C 180,E1 -9532.538,E2 -9532.538} C_VEL
LIN {X 0,Y 432.475,Z 419.324,A -85,B 0,C 180,E1 -9534.405,E2 -9534.405} C_VEL
LIN {X 0,Y 432.23,Z 421.645,A -85,B 0,C 180,E1 -9536.271,E2 -9536.271} C_VEL
LIN {X 0,Y 432.165,Z 422.593,A -85,B 0,C 180,E1 -9538.136,E2 -9538.136} C_VEL
LIN {X 0,Y 432.098,Z 422.206,A -85,B 0,C 180,E1 -9540,E2 -9540} C_VEL
LIN {X 0,Y 432.129,Z 420.48,A -85,B 0,C 180,E1 -9541.864,E2 -9541.864} C_VEL
LIN {X 0,Y 432.166,Z 417.403,A -85,B 0,C 180,E1 -9543.73,E2 -9543.73} C_VEL
LIN {X 0,Y 432.452,Z 412.863,A -85,B 0,C 180,E1 -9545.596,E2 -9545.596} C_VEL
LIN {X 0,Y 432.916,Z 406.732,A -85,B 0,C 180,E1 -9547.463,E2 -9547.463} C_VEL
LIN {X 0,Y 433.293,Z 399.876,A -85,B 0,C 180,E1 -9549.1,E2 -9549.1} C_VEL
LIN {X 0,Y 433.855,Z 391.356,A -85,B 0,C 180,E1 -9550.737,E2 -9550.737} C_VEL
LIN {X 0,Y 434.404,Z 382.5,A -85,B 0,C 180,E1 -9552.141,E2 -9552.141} C_VEL
LIN {X 0,Y 435.052,Z 373.752,A -85,B 0,C 180,E1 -9553.309,E2 -9553.309} C_VEL
LIN {X 0,Y 435.754,Z 362.905,A -85,B 0,C 180,E1 -9554.525,E2 -9554.525} C_VEL
LIN {X 0,Y 436.423,Z 350.776,A -85,B 0,C 180,E1 -9555.649,E2 -9555.649} C_VEL
LIN {X 0,Y 437.141,Z 338.374,A -85,B 0,C 180,E1 -9556.581,E2 -9556.581} C_VEL
LIN {X 0,Y 437.04,Z 334.862,A -85,B 0,C 180,E1 -9556.826,E2 -9556.826} C_VEL
LIN {X 0,Y 432.49,Z 319.777,A -85,B 0,C 180,E1 -9557.926,E2 -9557.926} C_VEL
LIN {X 0,Y 432.4,Z 319.279,A -85,B 0,C 180,E1 -9558.111,E2 -9558.111} C_VEL
LIN {X 0,Y 432.355,Z 319.257,A -85,B 0,C 180,E1 -9560.954,E2 -9560.954} C_VEL
LIN {X 0,Y 432.388,Z 319.252,A -85,B 0,C 180,E1 -9564.463,E2 -9564.463} C_VEL
LIN {X 0,Y 432.396,Z 319.248,A -85,B 0,C 180,E1 -9567.072,E2 -9567.072} C_VEL
LIN {X 0,Y 432.352,Z 319.256,A -85,B 0,C 180,E1 -9570.51,E2 -9570.51} C_VEL
LIN {X 0,Y 432.365,Z 319.25,A -85,B 0,C 180,E1 -9574.004,E2 -9574.004} C_VEL
LIN {X 0,Y 432.328,Z 319.254,A -85,B 0,C 180,E1 -9577.197,E2 -9577.197} C_VEL
LIN {X 0,Y 432.33,Z 319.26,A -85,B 0,C 180,E1 -9580.561,E2 -9580.561} C_VEL
LIN {X 0,Y 432.322,Z 319.255,A -85,B 0,C 180,E1 -9583.061,E2 -9583.061} C_VEL
LIN {X 0,Y 432.346,Z 319.251,A -85,B 0,C 180,E1 -9585.664,E2 -9585.664} C_VEL
LIN {X 0,Y 432.368,Z 319.256,A -85,B 0,C 180,E1 -9588.393,E2 -9588.393} C_VEL
LIN {X 0,Y 432.352,Z 319.252,A -85,B 0,C 180,E1 -9591.851,E2 -9591.851} C_VEL
LIN {X 0,Y 432.345,Z 319.251,A -85,B 0,C 180,E1 -9595.323,E2 -9595.323} C_VEL
LIN {X 0,Y 432.327,Z 319.256,A -85,B 0,C 180,E1 -9598.654,E2 -9598.654} C_VEL
LIN {X 0,Y 432.389,Z 319.249,A -85,B 0,C 180,E1 -9601.876,E2 -9601.876} C_VEL
LIN {X 0,Y 432.352,Z 319.25,A -85,B 0,C 180,E1 -9604.998,E2 -9604.998} C_VEL
LIN {X 0,Y 432.364,Z 319.256,A -85,B 0,C 180,E1 -9608.045,E2 -9608.045} C_VEL
LIN {X 0,Y 432.393,Z 319.245,A -85,B 0,C 180,E1 -9611.029,E2 -9611.029} C_VEL
LIN {X 0,Y 432.437,Z 319.247,A -85,B 0,C 180,E1 -9613.961,E2 -9613.961} C_VEL
LIN {X 0,Y 432.465,Z 319.242,A -85,B 0,C 180,E1 -9617.803,E2 -9617.803} C_VEL
LIN {X 0,Y 432.498,Z 319.236,A -85,B 0,C 180,E1 -9621.59,E2 -9621.59} C_VEL
LIN {X 0,Y 432.599,Z 319.221,A -85,B 0,C 180,E1 -9624.405,E2 -9624.405} C_VEL
LIN {X 0,Y 432.609,Z 319.221,A -85,B 0,C 180,E1 -9628.137,E2 -9628.137} C_VEL
LIN {X 0,Y 432.725,Z 319.207,A -85,B 0,C 180,E1 -9630.052,E2 -9630.052} C_VEL
LIN {X 0,Y 431.912,Z 319.305,A -85,B 0,C 180,E1 -9630.829,E2 -9630.829} C_VEL
LIN {X 0,Y 428.907,Z 319.682,A -85,B 0,C 180,E1 -9632.088,E2 -9632.088} C_VEL
LIN {X 0,Y 426.447,Z 319.991,A -85,B 0,C 180,E1 -9633.105,E2 -9633.105} C_VEL
LIN {X 0,Y 425.414,Z 320.119,A -85,B 0,C 180,E1 -9633.893,E2 -9633.893} C_VEL
LIN {X 0,Y 425.337,Z 320.126,A -85,B 0,C 180,E1 -9634.159,E2 -9634.159} C_VEL
LIN {X 0,Y 425.535,Z 320.099,A -85,B 0,C 180,E1 -9636.638,E2 -9636.638} C_VEL
LIN {X 0,Y 425.405,Z 320.122,A -85,B 0,C 180,E1 -9639.508,E2 -9639.508} C_VEL
LIN {X 0,Y 425.397,Z 320.117,A -85,B 0,C 180,E1 -9642.903,E2 -9642.903} C_VEL
LIN {X 0,Y 425.364,Z 320.121,A -85,B 0,C 180,E1 -9646.604,E2 -9646.604} C_VEL
LIN {X 0,Y 425.331,Z 320.13,A -85,B 0,C 180,E1 -9649.635,E2 -9649.635} C_VEL
LIN {X 0,Y 425.309,Z 320.135,A -85,B 0,C 180,E1 -9653.364,E2 -9653.364} C_VEL
LIN {X 0,Y 425.349,Z 320.124,A -85,B 0,C 180,E1 -9656.843,E2 -9656.843} C_VEL
LIN {X 0,Y 425.291,Z 320.132,A -85,B 0,C 180,E1 -9659.718,E2 -9659.718} C_VEL
LIN {X 0,Y 425.281,Z 320.136,A -85,B 0,C 180,E1 -9663.047,E2 -9663.047} C_VEL
LIN {X 0,Y 425.281,Z 320.132,A -85,B 0,C 180,E1 -9665.928,E2 -9665.928} C_VEL
LIN {X 0,Y 425.296,Z 320.135,A -85,B 0,C 180,E1 -9669.042,E2 -9669.042} C_VEL
LIN {X 0,Y 425.275,Z 320.134,A -85,B 0,C 180,E1 -9672.651,E2 -9672.651} C_VEL
LIN {X 0,Y 425.265,Z 320.133,A -85,B 0,C 180,E1 -9676.044,E2 -9676.044} C_VEL
LIN {X 0,Y 425.28,Z 320.133,A -85,B 0,C 180,E1 -9679.478,E2 -9679.478} C_VEL
LIN {X 0,Y 425.281,Z 320.133,A -85,B 0,C 180,E1 -9682.486,E2 -9682.486} C_VEL
LIN {X 0,Y 425.303,Z 320.128,A -85,B 0,C 180,E1 -9685.816,E2 -9685.816} C_VEL
LIN {X 0,Y 425.3,Z 320.131,A -85,B 0,C 180,E1 -9689.234,E2 -9689.234} C_VEL
LIN {X 0,Y 425.345,Z 320.126,A -85,B 0,C 180,E1 -9692.442,E2 -9692.442} C_VEL
LIN {X 0,Y 425.345,Z 320.123,A -85,B 0,C 180,E1 -9695.601,E2 -9695.601} C_VEL
LIN {X 0,Y 425.287,Z 320.138,A -85,B 0,C 180,E1 -9698.681,E2 -9698.681} C_VEL
LIN {X 0,Y 425.326,Z 320.125,A -85,B 0,C 180,E1 -9701.702,E2 -9701.702} C_VEL
LIN {X 0,Y 425.342,Z 320.13,A -85,B 0,C 180,E1 -9704.67,E2 -9704.67} C_VEL
LIN {X 0,Y 425.404,Z 320.116,A -85,B 0,C 180,E1 -9707.598,E2 -9707.598} C_VEL
LIN {X 0,Y 425.435,Z 320.112,A -85,B 0,C 180,E1 -9711.449,E2 -9711.449} C_VEL
LIN {X 0,Y 425.547,Z 320.103,A -85,B 0,C 180,E1 -9714.313,E2 -9714.313} C_VEL
LIN {X 0,Y 425.568,Z 320.099,A -85,B 0,C 180,E1 -9718.107,E2 -9718.107} C_VEL
LIN {X 0,Y 425.695,Z 320.082,A -85,B 0,C 180,E1 -9720,E2 -9720} C_VEL
LIN {X 0,Y 425.55,Z 320.099,A -85,B 0,C 180,E1 -9722.84,E2 -9722.84} C_VEL
LIN {X 0,Y 425.523,Z 320.104,A -85,B 0,C 180,E1 -9726.639,E2 -9726.639} C_VEL
LIN {X 0,Y 425.395,Z 320.117,A -85,B 0,C 180,E1 -9729.509,E2 -9729.509} C_VEL
LIN {X 0,Y 425.396,Z 320.117,A -85,B 0,C 180,E1 -9732.91,E2 -9732.91} C_VEL
LIN {X 0,Y 425.362,Z 320.123,A -85,B 0,C 180,E1 -9736.609,E2 -9736.609} C_VEL
LIN {X 0,Y 425.32,Z 320.128,A -85,B 0,C 180,E1 -9739.636,E2 -9739.636} C_VEL
LIN {X 0,Y 425.299,Z 320.13,A -85,B 0,C 180,E1 -9743.365,E2 -9743.365} C_VEL
LIN {X 0,Y 425.34,Z 320.124,A -85,B 0,C 180,E1 -9746.845,E2 -9746.845} C_VEL
LIN {X 0,Y 425.311,Z 320.132,A -85,B 0,C 180,E1 -9749.718,E2 -9749.718} C_VEL
LIN {X 0,Y 425.277,Z 320.132,A -85,B 0,C 180,E1 -9753.048,E2 -9753.048} C_VEL
LIN {X 0,Y 425.278,Z 320.138,A -85,B 0,C 180,E1 -9755.93,E2 -9755.93} C_VEL
LIN {X 0,Y 425.307,Z 320.132,A -85,B 0,C 180,E1 -9759.047,E2 -9759.047} C_VEL
LIN {X 0,Y 425.309,Z 320.135,A -85,B 0,C 180,E1 -9761.963,E2 -9761.963} C_VEL
LIN {X 0,Y 425.277,Z 320.292,A -85,B 0,C 180,E1 -9763.355,E2 -9763.355} C_VEL
LIN {X 0,Y 427.138,Z 329.087,A -85,B 0,C 180,E1 -9766.383,E2 -9766.383} C_VEL
LIN {X 0,Y 428.996,Z 338.184,A -85,B 0,C 180,E1 -9769.37,E2 -9769.37} C_VEL
LIN {X 0,Y 429.43,Z 342.279,A -85,B 0,C 180,E1 -9770.642,E2 -9770.642} C_VEL
LIN {X 0,Y 428.572,Z 351.964,A -85,B 0,C 180,E1 -9773.469,E2 -9773.469} C_VEL
LIN {X 0,Y 427.69,Z 362.801,A -85,B 0,C 180,E1 -9776.547,E2 -9776.547} C_VEL
LIN {X 0,Y 427.012,Z 374.732,A -85,B 0,C 180,E1 -9779.87,E2 -9779.87} C_VEL
LIN {X 0,Y 426.211,Z 388.358,A -85,B 0,C 180,E1 -9783.564,E2 -9783.564} C_VEL
LIN {X 0,Y 425.736,Z 399.987,A -85,B 0,C 180,E1 -9786.661,E2 -9786.661} C_VEL
LIN {X 0,Y 425.261,Z 411.52,A -85,B 0,C 180,E1 -9789.631,E2 -9789.631} C_VEL
LIN {X 0,Y 426.119,Z 418.015,A -85,B 0,C 180,E1 -9789.868,E2 -9789.868} C_VEL
LIN {X 0,Y 428.151,Z 433.186,A -85,B 0,C 180,E1 -9790.442,E2 -9790.442} C_VEL
LIN {X 0,Y 429.588,Z 447.33,A -85,B 0,C 180,E1 -9791.15,E2 -9791.15} C_VEL
LIN {X 0,Y 428.867,Z 460.806,A -85,B 0,C 180,E1 -9791.952,E2 -9791.952} C_VEL
LIN {X 0,Y 427.953,Z 473.838,A -85,B 0,C 180,E1 -9792.93,E2 -9792.93} C_VEL
LIN {X 0,Y 426.956,Z 486.615,A -85,B 0,C 180,E1 -9794.119,E2 -9794.119} C_VEL
LIN {X 0,Y 426.122,Z 498.151,A -85,B 0,C 180,E1 -9795.434,E2 -9795.434} C_VEL
LIN {X 0,Y 425.531,Z 508.066,A -85,B 0,C 180,E1 -9796.801,E2 -9796.801} C_VEL
LIN {X 0,Y 425.053,Z 517.164,A -85,B 0,C 180,E1 -9798.315,E2 -9798.315} C_VEL
LIN {X 0,Y 424.748,Z 524.342,A -85,B 0,C 180,E1 -9799.755,E2 -9799.755} C_VEL
LIN {X 0,Y 424.615,Z 531.194,A -85,B 0,C 180,E1 -9801.434,E2 -9801.434} C_VEL
LIN {X 0,Y 424.61,Z 537.007,A -85,B 0,C 180,E1 -9803.265,E2 -9803.265} C_VEL
LIN {X 0,Y 424.612,Z 539.601,A -85,B 0,C 180,E1 -9804.301,E2 -9804.301} C_VEL
LIN {X 0,Y 424.695,Z 543.167,A -85,B 0,C 180,E1 -9806.206,E2 -9806.206} C_VEL
LIN {X 0,Y 424.711,Z 545.209,A -85,B 0,C 180,E1 -9808.104,E2 -9808.104} C_VEL
LIN {X 0,Y 424.903,Z 545.81,A -85,B 0,C 180,E1 -9810.001,E2 -9810.001} C_VEL
LIN {X 0,Y 424.923,Z 545.551,A -85,B 0,C 180,E1 -9810.949,E2 -9810.949} C_VEL
LIN {X 0,Y 424.758,Z 543.9,A -85,B 0,C 180,E1 -9812.846,E2 -9812.846} C_VEL
LIN {X 0,Y 424.8,Z 540.763,A -85,B 0,C 180,E1 -9814.746,E2 -9814.746} C_VEL
LIN {X 0,Y 424.697,Z 536.024,A -85,B 0,C 180,E1 -9816.653,E2 -9816.653} C_VEL
LIN {X 0,Y 424.681,Z 531.397,A -85,B 0,C 180,E1 -9818.087,E2 -9818.087} C_VEL
LIN {X 0,Y 424.741,Z 524.659,A -85,B 0,C 180,E1 -9819.765,E2 -9819.765} C_VEL
LIN {X 0,Y 424.985,Z 516.324,A -85,B 0,C 180,E1 -9821.447,E2 -9821.447} C_VEL
LIN {X 0,Y 425.468,Z 506.103,A -85,B 0,C 180,E1 -9823.133,E2 -9823.133} C_VEL
LIN {X 0,Y 426.058,Z 495.601,A -85,B 0,C 180,E1 -9824.57,E2 -9824.57} C_VEL
LIN {X 0,Y 426.905,Z 484.112,A -85,B 0,C 180,E1 -9825.885,E2 -9825.885} C_VEL
LIN {X 0,Y 427.719,Z 471.605,A -85,B 0,C 180,E1 -9827.081,E2 -9827.081} C_VEL
LIN {X 0,Y 428.894,Z 457.959,A -85,B 0,C 180,E1 -9828.141,E2 -9828.141} C_VEL
LIN {X 0,Y 429.505,Z 446.993,A -85,B 0,C 180,E1 -9828.855,E2 -9828.855} C_VEL
LIN {X 0,Y 428.719,Z 434.654,A -85,B 0,C 180,E1 -9829.584,E2 -9829.584} C_VEL
LIN {X 0,Y 427.769,Z 419.932,A -85,B 0,C 180,E1 -9830.296,E2 -9830.296} C_VEL
LIN {X 0,Y 426.025,Z 407.453,A -85,B 0,C 180,E1 -9830.823,E2 -9830.823} C_VEL
LIN {X 0,Y 425.065,Z 401.664,A -85,B 0,C 180,E1 -9831.087,E2 -9831.087} C_VEL
LIN {X 0,Y 425.078,Z 398.543,A -85,B 0,C 180,E1 -9831.777,E2 -9831.777} C_VEL
LIN {X 0,Y 425.356,Z 385.527,A -85,B 0,C 180,E1 -9834.999,E2 -9834.999} C_VEL
LIN {X 0,Y 425.738,Z 371.447,A -85,B 0,C 180,E1 -9838.603,E2 -9838.603} C_VEL
LIN {X 0,Y 426.116,Z 359.338,A -85,B 0,C 180,E1 -9841.856,E2 -9841.856} C_VEL
LIN {X 0,Y 426.732,Z 347.666,A -85,B 0,C 180,E1 -9845.2,E2 -9845.2} C_VEL
LIN {X 0,Y 428.027,Z 336.739,A -85,B 0,C 180,E1 -9848.605,E2 -9848.605} C_VEL
LIN {X 0,Y 427.95,Z 333.282,A -85,B 0,C 180,E1 -9849.828,E2 -9849.828} C_VEL
LIN {X 0,Y 426.702,Z 326.821,A -85,B 0,C 180,E1 -9852.477,E2 -9852.477} C_VEL
LIN {X 0,Y 425.551,Z 321.158,A -85,B 0,C 180,E1 -9855.248,E2 -9855.248} C_VEL
LIN {X 0,Y 425.293,Z 320.174,A -85,B 0,C 180,E1 -9855.841,E2 -9855.841} C_VEL
LIN {X 0,Y 425.307,Z 320.133,A -85,B 0,C 180,E1 -9858.625,E2 -9858.625} C_VEL
LIN {X 0,Y 425.327,Z 320.131,A -85,B 0,C 180,E1 -9861.105,E2 -9861.105} C_VEL
LIN {X 0,Y 425.304,Z 320.131,A -85,B 0,C 180,E1 -9864.665,E2 -9864.665} C_VEL
LIN {X 0,Y 425.268,Z 320.137,A -85,B 0,C 180,E1 -9868.073,E2 -9868.073} C_VEL
LIN {X 0,Y 425.334,Z 320.13,A -85,B 0,C 180,E1 -9871.368,E2 -9871.368} C_VEL
LIN {X 0,Y 425.299,Z 320.134,A -85,B 0,C 180,E1 -9874.555,E2 -9874.555} C_VEL
LIN {X 0,Y 425.291,Z 320.137,A -85,B 0,C 180,E1 -9877.662,E2 -9877.662} C_VEL
LIN {X 0,Y 425.328,Z 320.32,A -85,B 0,C 180,E1 -9878.62,E2 -9878.62} C_VEL
LIN {X 0,Y 425.602,Z 321.493,A -85,B 0,C 180,E1 -9878.812,E2 -9878.812} C_VEL
LIN {X 0,Y 430.491,Z 333.343,A -85,B 0,C 180,E1 -9879.84,E2 -9879.84} C_VEL
LIN {X 0,Y 432.357,Z 339.185,A -85,B 0,C 180,E1 -9880.354,E2 -9880.354} C_VEL
LIN {X 0,Y 432.329,Z 343.306,A -85,B 0,C 180,E1 -9880.652,E2 -9880.652} C_VEL
LIN {X 0,Y 431.542,Z 355.53,A -85,B 0,C 180,E1 -9881.607,E2 -9881.607} C_VEL
LIN {X 0,Y 430.671,Z 366.698,A -85,B 0,C 180,E1 -9882.674,E2 -9882.674} C_VEL
LIN {X 0,Y 429.799,Z 376.965,A -85,B 0,C 180,E1 -9883.86,E2 -9883.86} C_VEL
LIN {X 0,Y 428.812,Z 387.573,A -85,B 0,C 180,E1 -9885.353,E2 -9885.353} C_VEL
LIN {X 0,Y 428.029,Z 395.54,A -85,B 0,C 180,E1 -9886.711,E2 -9886.711} C_VEL
LIN {X 0,Y 427.231,Z 403.565,A -85,B 0,C 180,E1 -9888.375,E2 -9888.375} C_VEL
LIN {X 0,Y 426.63,Z 409.967,A -85,B 0,C 180,E1 -9890.04,E2 -9890.04} C_VEL
LIN {X 0,Y 426.16,Z 414.96,A -85,B 0,C 180,E1 -9891.688,E2 -9891.688} C_VEL
LIN {X 0,Y 425.783,Z 418.803,A -85,B 0,C 180,E1 -9893.365,E2 -9893.365} C_VEL
LIN {X 0,Y 425.348,Z 421.8,A -85,B 0,C 180,E1 -9895.261,E2 -9895.261} C_VEL
LIN {X 0,Y 425.209,Z 423.389,A -85,B 0,C 180,E1 -9897.158,E2 -9897.158} C_VEL
LIN {X 0,Y 425.129,Z 423.623,A -85,B 0,C 180,E1 -9899.053,E2 -9899.053} C_VEL
LIN {X 0,Y 425.024,Z 422.534,A -85,B 0,C 180,E1 -9900.948,E2 -9900.948} C_VEL
LIN {X 0,Y 425.108,Z 421.472,A -85,B 0,C 180,E1 -9901.895,E2 -9901.895} C_VEL
LIN {X 0,Y 425.145,Z 418.348,A -85,B 0,C 180,E1 -9903.792,E2 -9903.792} C_VEL
LIN {X 0,Y 425.457,Z 413.754,A -85,B 0,C 180,E1 -9905.688,E2 -9905.688} C_VEL
LIN {X 0,Y 425.947,Z 407.566,A -85,B 0,C 180,E1 -9907.585,E2 -9907.585} C_VEL
LIN {X 0,Y 426.346,Z 400.642,A -85,B 0,C 180,E1 -9909.249,E2 -9909.249} C_VEL
LIN {X 0,Y 426.911,Z 392.059,A -85,B 0,C 180,E1 -9910.913,E2 -9910.913} C_VEL
LIN {X 0,Y 427.505,Z 383.134,A -85,B 0,C 180,E1 -9912.34,E2 -9912.34} C_VEL
LIN {X 0,Y 428.188,Z 374.315,A -85,B 0,C 180,E1 -9913.527,E2 -9913.527} C_VEL
LIN {X 0,Y 428.924,Z 362.826,A -85,B 0,C 180,E1 -9914.82,E2 -9914.82} C_VEL
LIN {X 0,Y 429.595,Z 351.171,A -85,B 0,C 180,E1 -9915.904,E2 -9915.904} C_VEL
LIN {X 0,Y 430.35,Z 338.667,A -85,B 0,C 180,E1 -9916.851,E2 -9916.851} C_VEL
LIN {X 0,Y 430.319,Z 336.958,A -85,B 0,C 180,E1 -9916.974,E2 -9916.974} C_VEL
LIN {X 0,Y 426.548,Z 324.269,A -85,B 0,C 180,E1 -9917.909,E2 -9917.909} C_VEL
LIN {X 0,Y 425.465,Z 320.811,A -85,B 0,C 180,E1 -9918.168,E2 -9918.168} C_VEL
LIN {X 0,Y 425.371,Z 320.159,A -85,B 0,C 180,E1 -9918.358,E2 -9918.358} C_VEL
LIN {X 0,Y 425.298,Z 320.134,A -85,B 0,C 180,E1 -9921.319,E2 -9921.319} C_VEL
LIN {X 0,Y 425.331,Z 320.132,A -85,B 0,C 180,E1 -9924.659,E2 -9924.659} C_VEL
LIN {X 0,Y 425.354,Z 320.122,A -85,B 0,C 180,E1 -9927.558,E2 -9927.558} C_VEL
LIN {X 0,Y 425.293,Z 320.135,A -85,B 0,C 180,E1 -9930.816,E2 -9930.816} C_VEL
LIN {X 0,Y 425.317,Z 320.13,A -85,B 0,C 180,E1 -9934.288,E2 -9934.288} C_VEL
LIN {X 0,Y 425.284,Z 320.131,A -85,B 0,C 180,E1 -9937.694,E2 -9937.694} C_VEL
LIN {X 0,Y 425.285,Z 320.138,A -85,B 0,C 180,E1 -9940.52,E2 -9940.52} C_VEL
LIN {X 0,Y 425.262,Z 320.133,A -85,B 0,C 180,E1 -9943.351,E2 -9943.351} C_VEL
LIN {X 0,Y 425.27,Z 320.137,A -85,B 0,C 180,E1 -9946.648,E2 -9946.648} C_VEL
LIN {X 0,Y 425.29,Z 320.13,A -85,B 0,C 180,E1 -9949.479,E2 -9949.479} C_VEL
LIN {X 0,Y 425.288,Z 320.135,A -85,B 0,C 180,E1 -9952.487,E2 -9952.487} C_VEL
LIN {X 0,Y 425.313,Z 320.129,A -85,B 0,C 180,E1 -9955.817,E2 -9955.817} C_VEL
LIN {X 0,Y 425.296,Z 320.129,A -85,B 0,C 180,E1 -9959.239,E2 -9959.239} C_VEL
LIN {X 0,Y 425.355,Z 320.126,A -85,B 0,C 180,E1 -9962.442,E2 -9962.442} C_VEL
LIN {X 0,Y 425.354,Z 320.124,A -85,B 0,C 180,E1 -9965.602,E2 -9965.602} C_VEL
LIN {X 0,Y 425.299,Z 320.13,A -85,B 0,C 180,E1 -9968.681,E2 -9968.681} C_VEL
LIN {X 0,Y 425.34,Z 320.127,A -85,B 0,C 180,E1 -9971.702,E2 -9971.702} C_VEL
LIN {X 0,Y 425.354,Z 320.122,A -85,B 0,C 180,E1 -9974.67,E2 -9974.67} C_VEL
LIN {X 0,Y 425.418,Z 320.117,A -85,B 0,C 180,E1 -9977.598,E2 -9977.598} C_VEL
LIN {X 0,Y 425.448,Z 320.113,A -85,B 0,C 180,E1 -9981.449,E2 -9981.449} C_VEL
LIN {X 0,Y 425.556,Z 320.099,A -85,B 0,C 180,E1 -9984.312,E2 -9984.312} C_VEL
LIN {X 0,Y 425.578,Z 320.097,A -85,B 0,C 180,E1 -9988.106,E2 -9988.106} C_VEL
LIN {X 0,Y 425.701,Z 320.083,A -85,B 0,C 180,E1 -9990.022,E2 -9990.022} C_VEL
LIN {X 0,Y 425.551,Z 320.097,A -85,B 0,C 180,E1 -9992.839,E2 -9992.839} C_VEL
LIN {X 0,Y 425.337,Z 320.126,A -85,B 0,C 180,E1 -9994.159,E2 -9994.159} C_VEL
LIN {X 0,Y 424.717,Z 320.203,A -85,B 0,C 180,E1 -9994.951,E2 -9994.951} C_VEL
LIN {X 0,Y 421.967,Z 320.545,A -85,B 0,C 180,E1 -9996.239,E2 -9996.239} C_VEL
LIN {X 0,Y 419.598,Z 320.842,A -85,B 0,C 180,E1 -9997.279,E2 -9997.279} C_VEL
LIN {X 0,Y 418.542,Z 320.973,A -85,B 0,C 180,E1 -9998.081,E2 -9998.081} C_VEL
LIN {X 0,Y 418.435,Z 320.984,A -85,B 0,C 180,E1 -9998.353,E2 -9998.353} C_VEL
LIN {X 0,Y 418.32,Z 321.005,A -85,B 0,C 180,E1 -10001.63,E2 -10001.63} C_VEL
LIN {X 0,Y 418.306,Z 321,A -85,B 0,C 180,E1 -10004.596,E2 -10004.596} C_VEL
LIN {X 0,Y 418.291,Z 321.008,A -85,B 0,C 180,E1 -10007.603,E2 -10007.603} C_VEL
LIN {X 0,Y 418.252,Z 321.007,A -85,B 0,C 180,E1 -10010.662,E2 -10010.662} C_VEL
LIN {X 0,Y 418.29,Z 321.005,A -85,B 0,C 180,E1 -10013.78,E2 -10013.78} C_VEL
LIN {X 0,Y 418.31,Z 321.003,A -85,B 0,C 180,E1 -10017.069,E2 -10017.069} C_VEL
LIN {X 0,Y 418.244,Z 321.007,A -85,B 0,C 180,E1 -10020.271,E2 -10020.271} C_VEL
LIN {X 0,Y 418.248,Z 321.009,A -85,B 0,C 180,E1 -10023.676,E2 -10023.676} C_VEL
LIN {X 0,Y 418.238,Z 321.015,A -85,B 0,C 180,E1 -10027.223,E2 -10027.223} C_VEL
LIN {X 0,Y 418.249,Z 321.009,A -85,B 0,C 180,E1 -10029.681,E2 -10029.681} C_VEL
LIN {X 0,Y 418.229,Z 321.01,A -85,B 0,C 180,E1 -10032.32,E2 -10032.32} C_VEL
LIN {X 0,Y 418.239,Z 321.015,A -85,B 0,C 180,E1 -10035.109,E2 -10035.109} C_VEL
LIN {X 0,Y 418.238,Z 321.009,A -85,B 0,C 180,E1 -10037.766,E2 -10037.766} C_VEL
LIN {X 0,Y 418.257,Z 321.009,A -85,B 0,C 180,E1 -10040.617,E2 -10040.617} C_VEL
LIN {X 0,Y 418.241,Z 321.008,A -85,B 0,C 180,E1 -10043.975,E2 -10043.975} C_VEL
LIN {X 0,Y 418.256,Z 321.01,A -85,B 0,C 180,E1 -10047.154,E2 -10047.154} C_VEL
LIN {X 0,Y 418.27,Z 321.012,A -85,B 0,C 180,E1 -10050.838,E2 -10050.838} C_VEL
LIN {X 0,Y 418.265,Z 321.006,A -85,B 0,C 180,E1 -10054.095,E2 -10054.095} C_VEL
LIN {X 0,Y 418.232,Z 321.011,A -85,B 0,C 180,E1 -10057.263,E2 -10057.263} C_VEL
LIN {X 0,Y 418.276,Z 321.007,A -85,B 0,C 180,E1 -10060.364,E2 -10060.364} C_VEL
LIN {X 0,Y 418.31,Z 321,A -85,B 0,C 180,E1 -10063.404,E2 -10063.404} C_VEL
LIN {X 0,Y 418.339,Z 320.998,A -85,B 0,C 180,E1 -10066.999,E2 -10066.999} C_VEL
LIN {X 0,Y 418.334,Z 321.001,A -85,B 0,C 180,E1 -10070.328,E2 -10070.328} C_VEL
LIN {X 0,Y 418.486,Z 320.978,A -85,B 0,C 180,E1 -10073.249,E2 -10073.249} C_VEL
LIN {X 0,Y 418.334,Z 320.997,A -85,B 0,C 180,E1 -10075.181,E2 -10075.181} C_VEL
LIN {X 0,Y 418.537,Z 320.974,A -85,B 0,C 180,E1 -10078.075,E2 -10078.075} C_VEL
LIN {X 0,Y 418.665,Z 320.958,A -85,B 0,C 180,E1 -10080,E2 -10080} C_VEL
LIN {X 0,Y 418.504,Z 320.977,A -85,B 0,C 180,E1 -10082.888,E2 -10082.888} C_VEL
LIN {X 0,Y 418.486,Z 320.98,A -85,B 0,C 180,E1 -10086.751,E2 -10086.751} C_VEL
LIN {X 0,Y 418.352,Z 320.996,A -85,B 0,C 180,E1 -10089.671,E2 -10089.671} C_VEL
LIN {X 0,Y 418.347,Z 320.995,A -85,B 0,C 180,E1 -10093.006,E2 -10093.006} C_VEL
LIN {X 0,Y 418.312,Z 321,A -85,B 0,C 180,E1 -10096.739,E2 -10096.739} C_VEL
LIN {X 0,Y 418.263,Z 321.009,A -85,B 0,C 180,E1 -10099.791,E2 -10099.791} C_VEL
LIN {X 0,Y 418.23,Z 321.01,A -85,B 0,C 180,E1 -10102.736,E2 -10102.736} C_VEL
LIN {X 0,Y 418.263,Z 321.012,A -85,B 0,C 180,E1 -10105.904,E2 -10105.904} C_VEL
LIN {X 0,Y 418.267,Z 321.005,A -85,B 0,C 180,E1 -10109.162,E2 -10109.162} C_VEL
LIN {X 0,Y 418.253,Z 321.006,A -85,B 0,C 180,E1 -10112.845,E2 -10112.845} C_VEL
LIN {X 0,Y 418.242,Z 321.014,A -85,B 0,C 180,E1 -10116.239,E2 -10116.239} C_VEL
LIN {X 0,Y 418.259,Z 321.013,A -85,B 0,C 180,E1 -10119.681,E2 -10119.681} C_VEL
LIN {X 0,Y 418.254,Z 321.115,A -85,B 0,C 180,E1 -10122.973,E2 -10122.973} C_VEL
LIN {X 0,Y 420.269,Z 330.788,A -85,B 0,C 180,E1 -10126.376,E2 -10126.376} C_VEL
LIN {X 0,Y 422.167,Z 340.247,A -85,B 0,C 180,E1 -10129.516,E2 -10129.516} C_VEL
LIN {X 0,Y 422.457,Z 344.303,A -85,B 0,C 180,E1 -10130.791,E2 -10130.791} C_VEL
LIN {X 0,Y 421.35,Z 356.158,A -85,B 0,C 180,E1 -10134.284,E2 -10134.284} C_VEL
LIN {X 0,Y 420.315,Z 369.633,A -85,B 0,C 180,E1 -10138.147,E2 -10138.147} C_VEL
LIN {X 0,Y 419.675,Z 379.618,A -85,B 0,C 180,E1 -10140.947,E2 -10140.947} C_VEL
LIN {X 0,Y 418.982,Z 392.921,A -85,B 0,C 180,E1 -10144.601,E2 -10144.601} C_VEL
LIN {X 0,Y 418.471,Z 403.543,A -85,B 0,C 180,E1 -10147.472,E2 -10147.472} C_VEL
LIN {X 0,Y 418.204,Z 410.711,A -85,B 0,C 180,E1 -10149.336,E2 -10149.336} C_VEL
LIN {X 0,Y 419.199,Z 418.37,A -85,B 0,C 180,E1 -10149.609,E2 -10149.609} C_VEL
LIN {X 0,Y 421.211,Z 433.544,A -85,B 0,C 180,E1 -10150.214,E2 -10150.214} C_VEL
LIN {X 0,Y 422.546,Z 447.627,A -85,B 0,C 180,E1 -10150.95,E2 -10150.95} C_VEL
LIN {X 0,Y 422.257,Z 455.845,A -85,B 0,C 180,E1 -10151.44,E2 -10151.44} C_VEL
LIN {X 0,Y 421.233,Z 469.617,A -85,B 0,C 180,E1 -10152.422,E2 -10152.422} C_VEL
LIN {X 0,Y 420.309,Z 481.593,A -85,B 0,C 180,E1 -10153.487,E2 -10153.487} C_VEL
LIN {X 0,Y 419.477,Z 492.846,A -85,B 0,C 180,E1 -10154.701,E2 -10154.701} C_VEL
LIN {X 0,Y 418.692,Z 503.959,A -85,B 0,C 180,E1 -10156.162,E2 -10156.162} C_VEL
LIN {X 0,Y 418.131,Z 513.174,A -85,B 0,C 180,E1 -10157.626,E2 -10157.626} C_VEL
LIN {X 0,Y 417.761,Z 522.008,A -85,B 0,C 180,E1 -10159.337,E2 -10159.337} C_VEL
LIN {X 0,Y 417.568,Z 528.202,A -85,B 0,C 180,E1 -10160.8,E2 -10160.8} C_VEL
LIN {X 0,Y 417.534,Z 533.313,A -85,B 0,C 180,E1 -10162.262,E2 -10162.262} C_VEL
LIN {X 0,Y 417.584,Z 536.932,A -85,B 0,C 180,E1 -10163.545,E2 -10163.545} C_VEL
LIN {X 0,Y 417.604,Z 540.503,A -85,B 0,C 180,E1 -10165.174,E2 -10165.174} C_VEL
LIN {X 0,Y 417.657,Z 542.103,A -85,B 0,C 180,E1 -10166.141,E2 -10166.141} C_VEL
LIN {X 0,Y 417.681,Z 544.16,A -85,B 0,C 180,E1 -10168.072,E2 -10168.072} C_VEL
LIN {X 0,Y 417.883,Z 544.771,A -85,B 0,C 180,E1 -10170.001,E2 -10170.001} C_VEL
LIN {X 0,Y 417.901,Z 544.512,A -85,B 0,C 180,E1 -10170.964,E2 -10170.964} C_VEL
LIN {X 0,Y 417.719,Z 542.863,A -85,B 0,C 180,E1 -10172.894,E2 -10172.894} C_VEL
LIN {X 0,Y 417.738,Z 541.491,A -85,B 0,C 180,E1 -10173.86,E2 -10173.86} C_VEL
LIN {X 0,Y 417.723,Z 538.674,A -85,B 0,C 180,E1 -10175.31,E2 -10175.31} C_VEL
LIN {X 0,Y 417.636,Z 533.55,A -85,B 0,C 180,E1 -10177.251,E2 -10177.251} C_VEL
LIN {X 0,Y 417.619,Z 528.541,A -85,B 0,C 180,E1 -10178.712,E2 -10178.712} C_VEL
LIN {X 0,Y 417.733,Z 521.381,A -85,B 0,C 180,E1 -10180.421,E2 -10180.421} C_VEL
LIN {X 0,Y 418.078,Z 512.593,A -85,B 0,C 180,E1 -10182.131,E2 -10182.131} C_VEL
LIN {X 0,Y 418.576,Z 503.527,A -85,B 0,C 180,E1 -10183.596,E2 -10183.596} C_VEL
LIN {X 0,Y 419.306,Z 491.759,A -85,B 0,C 180,E1 -10185.183,E2 -10185.183} C_VEL
LIN {X 0,Y 420.278,Z 479.757,A -85,B 0,C 180,E1 -10186.516,E2 -10186.516} C_VEL
LIN {X 0,Y 421.243,Z 467.405,A -85,B 0,C 180,E1 -10187.661,E2 -10187.661} C_VEL
LIN {X 0,Y 422.365,Z 454.02,A -85,B 0,C 180,E1 -10188.683,E2 -10188.683} C_VEL
LIN {X 0,Y 422.711,Z 448.582,A -85,B 0,C 180,E1 -10189.044,E2 -10189.044} C_VEL
LIN {X 0,Y 422.032,Z 436.424,A -85,B 0,C 180,E1 -10189.818,E2 -10189.818} C_VEL
LIN {X 0,Y 421.154,Z 420.779,A -85,B 0,C 180,E1 -10190.63,E2 -10190.63} C_VEL
LIN {X 0,Y 419.307,Z 407.133,A -85,B 0,C 180,E1 -10191.251,E2 -10191.251} C_VEL
LIN {X 0,Y 418.017,Z 400.17,A -85,B 0,C 180,E1 -10191.579,E2 -10191.579} C_VEL
LIN {X 0,Y 418.006,Z 399.271,A -85,B 0,C 180,E1 -10191.71,E2 -10191.71} C_VEL
LIN {X 0,Y 418.287,Z 386.77,A -85,B 0,C 180,E1 -10194.865,E2 -10194.865} C_VEL
LIN {X 0,Y 418.691,Z 372.541,A -85,B 0,C 180,E1 -10198.581,E2 -10198.581} C_VEL
LIN {X 0,Y 419.106,Z 360.511,A -85,B 0,C 180,E1 -10201.886,E2 -10201.886} C_VEL
LIN {X 0,Y 419.797,Z 348.901,A -85,B 0,C 180,E1 -10205.298,E2 -10205.298} C_VEL
LIN {X 0,Y 421.15,Z 338.079,A -85,B 0,C 180,E1 -10208.758,E2 -10208.758} C_VEL
LIN {X 0,Y 421.08,Z 335.081,A -85,B 0,C 180,E1 -10209.847,E2 -10209.847} C_VEL
LIN {X 0,Y 419.863,Z 328.582,A -85,B 0,C 180,E1 -10212.565,E2 -10212.565} C_VEL
LIN {X 0,Y 418.781,Z 323.331,A -85,B 0,C 180,E1 -10215.183,E2 -10215.183} C_VEL
LIN {X 0,Y 418.217,Z 321.036,A -85,B 0,C 180,E1 -10216.614,E2 -10216.614} C_VEL
LIN {X 0,Y 418.269,Z 321.011,A -85,B 0,C 180,E1 -10219.124,E2 -10219.124} C_VEL
LIN {X 0,Y 418.241,Z 321.013,A -85,B 0,C 180,E1 -10222.165,E2 -10222.165} C_VEL
LIN {X 0,Y 418.269,Z 321.01,A -85,B 0,C 180,E1 -10225.42,E2 -10225.42} C_VEL
LIN {X 0,Y 418.214,Z 321.015,A -85,B 0,C 180,E1 -10228.604,E2 -10228.604} C_VEL
LIN {X 0,Y 418.295,Z 321.007,A -85,B 0,C 180,E1 -10231.937,E2 -10231.937} C_VEL
LIN {X 0,Y 418.293,Z 321.007,A -85,B 0,C 180,E1 -10235.163,E2 -10235.163} C_VEL
LIN {X 0,Y 418.305,Z 321.165,A -85,B 0,C 180,E1 -10238.093,E2 -10238.093} C_VEL
LIN {X 0,Y 418.55,Z 322.256,A -85,B 0,C 180,E1 -10238.291,E2 -10238.291} C_VEL
LIN {X 0,Y 423.996,Z 335.26,A -85,B 0,C 180,E1 -10239.478,E2 -10239.478} C_VEL
LIN {X 0,Y 426.069,Z 341.84,A -85,B 0,C 180,E1 -10240.089,E2 -10240.089} C_VEL
LIN {X 0,Y 425.199,Z 354.647,A -85,B 0,C 180,E1 -10241.072,E2 -10241.072} C_VEL
LIN {X 0,Y 424.289,Z 366.119,A -85,B 0,C 180,E1 -10242.156,E2 -10242.156} C_VEL
LIN {X 0,Y 423.366,Z 376.644,A -85,B 0,C 180,E1 -10243.36,E2 -10243.36} C_VEL
LIN {X 0,Y 422.535,Z 385.473,A -85,B 0,C 180,E1 -10244.566,E2 -10244.566} C_VEL
LIN {X 0,Y 421.675,Z 392.993,A -85,B 0,C 180,E1 -10245.769,E2 -10245.769} C_VEL
LIN {X 0,Y 420.827,Z 401.714,A -85,B 0,C 180,E1 -10247.461,E2 -10247.461} C_VEL
LIN {X 0,Y 420.145,Z 407.805,A -85,B 0,C 180,E1 -10248.909,E2 -10248.909} C_VEL
LIN {X 0,Y 419.635,Z 412.814,A -85,B 0,C 180,E1 -10250.359,E2 -10250.359} C_VEL
LIN {X 0,Y 419.073,Z 417.995,A -85,B 0,C 180,E1 -10252.29,E2 -10252.29} C_VEL
LIN {X 0,Y 418.536,Z 421.668,A -85,B 0,C 180,E1 -10254.218,E2 -10254.218} C_VEL
LIN {X 0,Y 418.263,Z 423.907,A -85,B 0,C 180,E1 -10256.146,E2 -10256.146} C_VEL
LIN {X 0,Y 418.177,Z 424.757,A -85,B 0,C 180,E1 -10258.074,E2 -10258.074} C_VEL
LIN {X 0,Y 418.083,Z 424.279,A -85,B 0,C 180,E1 -10260,E2 -10260} C_VEL
LIN {X 0,Y 418.087,Z 422.462,A -85,B 0,C 180,E1 -10261.927,E2 -10261.927} C_VEL
LIN {X 0,Y 418.124,Z 419.286,A -85,B 0,C 180,E1 -10263.855,E2 -10263.855} C_VEL
LIN {X 0,Y 418.463,Z 414.632,A -85,B 0,C 180,E1 -10265.784,E2 -10265.784} C_VEL
LIN {X 0,Y 418.814,Z 410.077,A -85,B 0,C 180,E1 -10267.23,E2 -10267.23} C_VEL
LIN {X 0,Y 419.198,Z 403.515,A -85,B 0,C 180,E1 -10268.922,E2 -10268.922} C_VEL
LIN {X 0,Y 419.809,Z 395.384,A -85,B 0,C 180,E1 -10270.612,E2 -10270.612} C_VEL
LIN {X 0,Y 420.42,Z 386.916,A -85,B 0,C 180,E1 -10272.062,E2 -10272.062} C_VEL
LIN {X 0,Y 421.094,Z 376.76,A -85,B 0,C 180,E1 -10273.513,E2 -10273.513} C_VEL
LIN {X 0,Y 421.931,Z 366.093,A -85,B 0,C 180,E1 -10274.77,E2 -10274.77} C_VEL
LIN {X 0,Y 422.649,Z 354.299,A -85,B 0,C 180,E1 -10275.925,E2 -10275.925} C_VEL
LIN {X 0,Y 423.372,Z 342.297,A -85,B 0,C 180,E1 -10276.888,E2 -10276.888} C_VEL
LIN {X 0,Y 423.523,Z 338.876,A -85,B 0,C 180,E1 -10277.131,E2 -10277.131} C_VEL
LIN {X 0,Y 419.951,Z 326.624,A -85,B 0,C 180,E1 -10278.066,E2 -10278.066} C_VEL
LIN {X 0,Y 418.45,Z 321.774,A -85,B 0,C 180,E1 -10278.419,E2 -10278.419} C_VEL
LIN {X 0,Y 418.324,Z 321.039,A -85,B 0,C 180,E1 -10278.615,E2 -10278.615} C_VEL
LIN {X 0,Y 418.239,Z 321.012,A -85,B 0,C 180,E1 -10281.696,E2 -10281.696} C_VEL
LIN {X 0,Y 418.289,Z 321.008,A -85,B 0,C 180,E1 -10284.865,E2 -10284.865} C_VEL
LIN {X 0,Y 418.296,Z 321.002,A -85,B 0,C 180,E1 -10288.063,E2 -10288.063} C_VEL
LIN {X 0,Y 418.216,Z 321.011,A -85,B 0,C 180,E1 -10291.396,E2 -10291.396} C_VEL
LIN {X 0,Y 418.271,Z 321.012,A -85,B 0,C 180,E1 -10294.58,E2 -10294.58} C_VEL
LIN {X 0,Y 418.231,Z 321.01,A -85,B 0,C 180,E1 -10297.833,E2 -10297.833} C_VEL
LIN {X 0,Y 418.227,Z 321.012,A -85,B 0,C 180,E1 -10300.948,E2 -10300.948} C_VEL
LIN {X 0,Y 418.215,Z 321.012,A -85,B 0,C 180,E1 -10303.729,E2 -10303.729} C_VEL
LIN {X 0,Y 418.222,Z 321.017,A -85,B 0,C 180,E1 -10306.45,E2 -10306.45} C_VEL
LIN {X 0,Y 418.266,Z 321.005,A -85,B 0,C 180,E1 -10309.124,E2 -10309.124} C_VEL
LIN {X 0,Y 418.239,Z 321.014,A -85,B 0,C 180,E1 -10312.165,E2 -10312.165} C_VEL
LIN {X 0,Y 418.271,Z 321.004,A -85,B 0,C 180,E1 -10315.42,E2 -10315.42} C_VEL
LIN {X 0,Y 418.218,Z 321.014,A -85,B 0,C 180,E1 -10318.604,E2 -10318.604} C_VEL
LIN {X 0,Y 418.298,Z 321.005,A -85,B 0,C 180,E1 -10321.936,E2 -10321.936} C_VEL
LIN {X 0,Y 418.296,Z 321.001,A -85,B 0,C 180,E1 -10325.162,E2 -10325.162} C_VEL
LIN {X 0,Y 418.24,Z 321.013,A -85,B 0,C 180,E1 -10328.303,E2 -10328.303} C_VEL
LIN {X 0,Y 418.29,Z 321.003,A -85,B 0,C 180,E1 -10331.383,E2 -10331.383} C_VEL
LIN {X 0,Y 418.309,Z 321.002,A -85,B 0,C 180,E1 -10334.405,E2 -10334.405} C_VEL
LIN {X 0,Y 418.361,Z 320.994,A -85,B 0,C 180,E1 -10337.385,E2 -10337.385} C_VEL
LIN {X 0,Y 418.406,Z 320.989,A -85,B 0,C 180,E1 -10341.304,E2 -10341.304} C_VEL
LIN {X 0,Y 418.516,Z 320.977,A -85,B 0,C 180,E1 -10344.216,E2 -10344.216} C_VEL
LIN {X 0,Y 418.547,Z 320.973,A -85,B 0,C 180,E1 -10348.075,E2 -10348.075} C_VEL
LIN {X 0,Y 418.676,Z 320.958,A -85,B 0,C 180,E1 -10349.999,E2 -10349.999} C_VEL
LIN {X 0,Y 418.506,Z 320.975,A -85,B 0,C 180,E1 -10352.887,E2 -10352.887} C_VEL
LIN {X 0,Y 418.498,Z 320.976,A -85,B 0,C 180,E1 -10356.75,E2 -10356.75} C_VEL
LIN {X 0,Y 418.435,Z 320.984,A -85,B 0,C 180,E1 -10358.353,E2 -10358.353} C_VEL
LIN {X 0,Y 417.699,Z 321.08,A -85,B 0,C 180,E1 -10359.155,E2 -10359.155} C_VEL
LIN {X 0,Y 414.781,Z 321.439,A -85,B 0,C 180,E1 -10360.459,E2 -10360.459} C_VEL
LIN {X 0,Y 412.366,Z 321.747,A -85,B 0,C 180,E1 -10361.512,E2 -10361.512} C_VEL
LIN {X 0,Y 411.359,Z 321.866,A -85,B 0,C 180,E1 -10362.326,E2 -10362.326} C_VEL
LIN {X 0,Y 411.291,Z 321.874,A -85,B 0,C 180,E1 -10362.601,E2 -10362.601} C_VEL
LIN {X 0,Y 411.258,Z 321.881,A -85,B 0,C 180,E1 -10365.867,E2 -10365.867} C_VEL
LIN {X 0,Y 411.227,Z 321.883,A -85,B 0,C 180,E1 -10368.947,E2 -10368.947} C_VEL
LIN {X 0,Y 411.206,Z 321.885,A -85,B 0,C 180,E1 -10372.641,E2 -10372.641} C_VEL
LIN {X 0,Y 411.237,Z 321.887,A -85,B 0,C 180,E1 -10375.292,E2 -10375.292} C_VEL
LIN {X 0,Y 411.259,Z 321.883,A -85,B 0,C 180,E1 -10377.476,E2 -10377.476} C_VEL
LIN {X 0,Y 411.189,Z 321.889,A -85,B 0,C 180,E1 -10380.846,E2 -10380.846} C_VEL
LIN {X 0,Y 411.204,Z 321.885,A -85,B 0,C 180,E1 -10384.332,E2 -10384.332} C_VEL
LIN {X 0,Y 411.194,Z 321.886,A -85,B 0,C 180,E1 -10387.972,E2 -10387.972} C_VEL
LIN {X 0,Y 411.179,Z 321.889,A -85,B 0,C 180,E1 -10390.503,E2 -10390.503} C_VEL
LIN {X 0,Y 411.175,Z 321.895,A -85,B 0,C 180,E1 -10393.132,E2 -10393.132} C_VEL
LIN {X 0,Y 411.17,Z 321.889,A -85,B 0,C 180,E1 -10395.879,E2 -10395.879} C_VEL
LIN {X 0,Y 411.161,Z 321.894,A -85,B 0,C 180,E1 -10398.77,E2 -10398.77} C_VEL
LIN {X 0,Y 411.208,Z 321.884,A -85,B 0,C 180,E1 -10401.829,E2 -10401.829} C_VEL
LIN {X 0,Y 411.207,Z 321.889,A -85,B 0,C 180,E1 -10405.12,E2 -10405.12} C_VEL
LIN {X 0,Y 411.168,Z 321.889,A -85,B 0,C 180,E1 -10408.002,E2 -10408.002} C_VEL
LIN {X 0,Y 411.219,Z 321.884,A -85,B 0,C 180,E1 -10411.41,E2 -10411.41} C_VEL
LIN {X 0,Y 411.23,Z 321.888,A -85,B 0,C 180,E1 -10414.706,E2 -10414.706} C_VEL
LIN {X 0,Y 411.199,Z 321.885,A -85,B 0,C 180,E1 -10417.913,E2 -10417.913} C_VEL
LIN {X 0,Y 411.218,Z 321.886,A -85,B 0,C 180,E1 -10421.051,E2 -10421.051} C_VEL
LIN {X 0,Y 411.248,Z 321.881,A -85,B 0,C 180,E1 -10424.131,E2 -10424.131} C_VEL
LIN {X 0,Y 411.295,Z 321.874,A -85,B 0,C 180,E1 -10427.165,E2 -10427.165} C_VEL
LIN {X 0,Y 411.286,Z 321.877,A -85,B 0,C 180,E1 -10430.161,E2 -10430.161} C_VEL
LIN {X 0,Y 411.453,Z 321.854,A -85,B 0,C 180,E1 -10433.133,E2 -10433.133} C_VEL
LIN {X 0,Y 411.305,Z 321.873,A -85,B 0,C 180,E1 -10435.099,E2 -10435.099} C_VEL
LIN {X 0,Y 411.506,Z 321.85,A -85,B 0,C 180,E1 -10438.042,E2 -10438.042} C_VEL
LIN {X 0,Y 411.634,Z 321.834,A -85,B 0,C 180,E1 -10440,E2 -10440} C_VEL
LIN {X 0,Y 411.459,Z 321.854,A -85,B 0,C 180,E1 -10442.937,E2 -10442.937} C_VEL
LIN {X 0,Y 411.452,Z 321.855,A -85,B 0,C 180,E1 -10446.867,E2 -10446.867} C_VEL
LIN {X 0,Y 411.3,Z 321.875,A -85,B 0,C 180,E1 -10449.838,E2 -10449.838} C_VEL
LIN {X 0,Y 411.305,Z 321.872,A -85,B 0,C 180,E1 -10453.109,E2 -10453.109} C_VEL
LIN {X 0,Y 411.255,Z 321.879,A -85,B 0,C 180,E1 -10456.889,E2 -10456.889} C_VEL
LIN {X 0,Y 411.222,Z 321.888,A -85,B 0,C 180,E1 -10459.987,E2 -10459.987} C_VEL
LIN {X 0,Y 411.195,Z 321.886,A -85,B 0,C 180,E1 -10463.148,E2 -10463.148} C_VEL
LIN {X 0,Y 411.23,Z 321.884,A -85,B 0,C 180,E1 -10466.381,E2 -10466.381} C_VEL
LIN {X 0,Y 411.204,Z 321.889,A -85,B 0,C 180,E1 -10469.712,E2 -10469.712} C_VEL
LIN {X 0,Y 411.199,Z 321.886,A -85,B 0,C 180,E1 -10473.156,E2 -10473.156} C_VEL
LIN {X 0,Y 411.189,Z 321.89,A -85,B 0,C 180,E1 -10476.554,E2 -10476.554} C_VEL
LIN {X 0,Y 411.222,Z 321.89,A -85,B 0,C 180,E1 -10479.731,E2 -10479.731} C_VEL
LIN {X 0,Y 411.218,Z 322.051,A -85,B 0,C 180,E1 -10482.663,E2 -10482.663} C_VEL
LIN {X 0,Y 413.309,Z 332.204,A -85,B 0,C 180,E1 -10486.275,E2 -10486.275} C_VEL
LIN {X 0,Y 414.986,Z 340.407,A -85,B 0,C 180,E1 -10489.055,E2 -10489.055} C_VEL
LIN {X 0,Y 415.511,Z 345.266,A -85,B 0,C 180,E1 -10490.621,E2 -10490.621} C_VEL
LIN {X 0,Y 414.279,Z 358.264,A -85,B 0,C 180,E1 -10494.517,E2 -10494.517} C_VEL
LIN {X 0,Y 413.257,Z 371.058,A -85,B 0,C 180,E1 -10498.246,E2 -10498.246} C_VEL
LIN {X 0,Y 412.62,Z 380.57,A -85,B 0,C 180,E1 -10500.961,E2 -10500.961} C_VEL
LIN {X 0,Y 411.876,Z 394.099,A -85,B 0,C 180,E1 -10504.75,E2 -10504.75} C_VEL
LIN {X 0,Y 411.295,Z 405.589,A -85,B 0,C 180,E1 -10507.92,E2 -10507.92} C_VEL
LIN {X 0,Y 411.143,Z 410.009,A -85,B 0,C 180,E1 -10509.045,E2 -10509.045} C_VEL
LIN {X 0,Y 413.634,Z 429.041,A -85,B 0,C 180,E1 -10509.763,E2 -10509.763} C_VEL
LIN {X 0,Y 415.1,Z 443.098,A -85,B 0,C 180,E1 -10510.466,E2 -10510.466} C_VEL
LIN {X 0,Y 415.604,Z 451.095,A -85,B 0,C 180,E1 -10510.94,E2 -10510.94} C_VEL
LIN {X 0,Y 414.699,Z 463.682,A -85,B 0,C 180,E1 -10511.786,E2 -10511.786} C_VEL
LIN {X 0,Y 413.77,Z 476.227,A -85,B 0,C 180,E1 -10512.836,E2 -10512.836} C_VEL
LIN {X 0,Y 412.769,Z 488.18,A -85,B 0,C 180,E1 -10514.066,E2 -10514.066} C_VEL
LIN {X 0,Y 411.92,Z 499.072,A -85,B 0,C 180,E1 -10515.425,E2 -10515.425} C_VEL
LIN {X 0,Y 411.281,Z 508.931,A -85,B 0,C 180,E1 -10516.911,E2 -10516.911} C_VEL
LIN {X 0,Y 410.863,Z 517.182,A -85,B 0,C 180,E1 -10518.406,E2 -10518.406} C_VEL
LIN {X 0,Y 410.578,Z 525.062,A -85,B 0,C 180,E1 -10520.145,E2 -10520.145} C_VEL
LIN {X 0,Y 410.483,Z 530.539,A -85,B 0,C 180,E1 -10521.633,E2 -10521.633} C_VEL
LIN {X 0,Y 410.538,Z 536.001,A -85,B 0,C 180,E1 -10523.512,E2 -10523.512} C_VEL
LIN {X 0,Y 410.562,Z 539.407,A -85,B 0,C 180,E1 -10525.091,E2 -10525.091} C_VEL
LIN {X 0,Y 410.619,Z 541.02,A -85,B 0,C 180,E1 -10526.075,E2 -10526.075} C_VEL
LIN {X 0,Y 410.652,Z 543.099,A -85,B 0,C 180,E1 -10528.039,E2 -10528.039} C_VEL
LIN {X 0,Y 410.862,Z 543.724,A -85,B 0,C 180,E1 -10530.001,E2 -10530.001} C_VEL
LIN {X 0,Y 410.877,Z 543.471,A -85,B 0,C 180,E1 -10530.981,E2 -10530.981} C_VEL
LIN {X 0,Y 410.681,Z 541.823,A -85,B 0,C 180,E1 -10532.944,E2 -10532.944} C_VEL
LIN {X 0,Y 410.701,Z 540.458,A -85,B 0,C 180,E1 -10533.926,E2 -10533.926} C_VEL
LIN {X 0,Y 410.651,Z 537.637,A -85,B 0,C 180,E1 -10535.402,E2 -10535.402} C_VEL
LIN {X 0,Y 410.574,Z 532.512,A -85,B 0,C 180,E1 -10537.377,E2 -10537.377} C_VEL
LIN {X 0,Y 410.535,Z 527.514,A -85,B 0,C 180,E1 -10538.864,E2 -10538.864} C_VEL
LIN {X 0,Y 410.696,Z 520.363,A -85,B 0,C 180,E1 -10540.601,E2 -10540.601} C_VEL
LIN {X 0,Y 411.016,Z 511.599,A -85,B 0,C 180,E1 -10542.342,E2 -10542.342} C_VEL
LIN {X 0,Y 411.557,Z 502.571,A -85,B 0,C 180,E1 -10543.833,E2 -10543.833} C_VEL
LIN {X 0,Y 412.287,Z 491.87,A -85,B 0,C 180,E1 -10545.321,E2 -10545.321} C_VEL
LIN {X 0,Y 413.289,Z 480.213,A -85,B 0,C 180,E1 -10546.677,E2 -10546.677} C_VEL
LIN {X 0,Y 414.225,Z 468.899,A -85,B 0,C 180,E1 -10547.783,E2 -10547.783} C_VEL
LIN {X 0,Y 415.475,Z 455.405,A -85,B 0,C 180,E1 -10548.876,E2 -10548.876} C_VEL
LIN {X 0,Y 415.824,Z 448.404,A -85,B 0,C 180,E1 -10549.372,E2 -10549.372} C_VEL
LIN {X 0,Y 415.272,Z 434.796,A -85,B 0,C 180,E1 -10550.262,E2 -10550.262} C_VEL
LIN {X 0,Y 414.393,Z 419.501,A -85,B 0,C 180,E1 -10551.089,E2 -10551.089} C_VEL
LIN {X 0,Y 412.57,Z 407.088,A -85,B 0,C 180,E1 -10551.702,E2 -10551.702} C_VEL
